LIN {X 0,Y 122.91,Z 344.93,A -85,B 0,C 180,E1 -26212.698,E2 -26212.698} C_VEL
LIN {X 0,Y 127.264,Z 335.4,A -85,B 0,C 180,E1 -26216.213,E2 -26216.213} C_VEL
LIN {X 0,Y 131.785,Z 325.121,A -85,B 0,C 180,E1 -26219.114,E2 -26219.114} C_VEL
LIN {X 0,Y 136.511,Z 312.597,A -85,B 0,C 180,E1 -26221.845,E2 -26221.845} C_VEL
LIN {X 0,Y 140.339,Z 300.53,A -85,B 0,C 180,E1 -26223.852,E2 -26223.852} C_VEL
LIN {X 0,Y 143.644,Z 287.351,A -85,B 0,C 180,E1 -26225.516,E2 -26225.516} C_VEL
LIN {X 0,Y 146.296,Z 273.12,A -85,B 0,C 180,E1 -26226.793,E2 -26226.793} C_VEL
LIN {X 0,Y 148.096,Z 259.317,A -85,B 0,C 180,E1 -26227.549,E2 -26227.549} C_VEL
LIN {X 0,Y 152.361,Z 207.795,A -85,B 0,C 180,E1 -26229.457,E2 -26229.457} C_VEL
LIN {X 0,Y 147.363,Z 196.9,A -85,B 0,C 180,E1 -26232.578,E2 -26232.578} C_VEL
LIN {X 0,Y 142.317,Z 187.434,A -85,B 0,C 180,E1 -26236.042,E2 -26236.042} C_VEL
LIN {X 0,Y 138.298,Z 180.817,A -85,B 0,C 180,E1 -26239.137,E2 -26239.137} C_VEL
LIN {X 0,Y 134.118,Z 174.322,A -85,B 0,C 180,E1 -26242.853,E2 -26242.853} C_VEL
LIN {X 0,Y 130.981,Z 169.962,A -85,B 0,C 180,E1 -26246.076,E2 -26246.076} C_VEL
LIN {X 0,Y 128.411,Z 166.477,A -85,B 0,C 180,E1 -26249.154,E2 -26249.154} C_VEL
LIN {X 0,Y 127.763,Z 165.521,A -85,B 0,C 180,E1 -26250.031,E2 -26250.031} C_VEL
LIN {X 0,Y 125.309,Z 162.834,A -85,B 0,C 180,E1 -26253.6,E2 -26253.6} C_VEL
LIN {X 0,Y 124.174,Z 160.568,A -85,B 0,C 180,E1 -26255.787,E2 -26255.787} C_VEL
LIN {X 0,Y 121.255,Z 158.023,A -85,B 0,C 180,E1 -26262.732,E2 -26262.732} C_VEL
LIN {X 0,Y 120.363,Z 155.046,A -85,B 0,C 180,E1 -26268.375,E2 -26268.375} C_VEL
LIN {X 0,Y 120.599,Z 154.855,A -85,B 0,C 180,E1 -26276.67,E2 -26276.67} C_VEL
LIN {X 0,Y 120.863,Z 155.058,A -85,B 0,C 180,E1 -26278.137,E2 -26278.137} C_VEL
LIN {X 0,Y 121.622,Z 157.801,A -85,B 0,C 180,E1 -26281.874,E2 -26281.874} C_VEL
LIN {X 0,Y 123.928,Z 160.174,A -85,B 0,C 180,E1 -26287.341,E2 -26287.341} C_VEL
LIN {X 0,Y 124.584,Z 160.744,A -85,B 0,C 180,E1 -26288.526,E2 -26288.526} C_VEL
LIN {X 0,Y 126.362,Z 163.972,A -85,B 0,C 180,E1 -26291.642,E2 -26291.642} C_VEL
LIN {X 0,Y 128.449,Z 166.176,A -85,B 0,C 180,E1 -26294.466,E2 -26294.466} C_VEL
LIN {X 0,Y 131.151,Z 169.964,A -85,B 0,C 180,E1 -26297.718,E2 -26297.718} C_VEL
LIN {X 0,Y 135.213,Z 176.102,A -85,B 0,C 180,E1 -26301.831,E2 -26301.831} C_VEL
LIN {X 0,Y 137.802,Z 180.05,A -85,B 0,C 180,E1 -26304.089,E2 -26304.089} C_VEL
LIN {X 0,Y 142.126,Z 187.185,A -85,B 0,C 180,E1 -26307.455,E2 -26307.455} C_VEL
LIN {X 0,Y 145.883,Z 194.238,A -85,B 0,C 180,E1 -26310.095,E2 -26310.095} C_VEL
LIN {X 0,Y 150.285,Z 206.436,A -85,B 0,C 180,E1 -26313.156,E2 -26313.156} C_VEL
LIN {X 0,Y 152.175,Z 212.724,A -85,B 0,C 180,E1 -26314.44,E2 -26314.44} C_VEL
LIN {X 0,Y 147.482,Z 269.48,A -85,B 0,C 180,E1 -26316.622,E2 -26316.622} C_VEL
LIN {X 0,Y 145.239,Z 284.153,A -85,B 0,C 180,E1 -26317.599,E2 -26317.599} C_VEL
LIN {X 0,Y 142.244,Z 297.61,A -85,B 0,C 180,E1 -26318.913,E2 -26318.913} C_VEL
LIN {X 0,Y 138.11,Z 311.658,A -85,B 0,C 180,E1 -26320.811,E2 -26320.811} C_VEL
LIN {X 0,Y 133.642,Z 324.22,A -85,B 0,C 180,E1 -26323.141,E2 -26323.141} C_VEL
LIN {X 0,Y 129.478,Z 334.557,A -85,B 0,C 180,E1 -26325.672,E2 -26325.672} C_VEL
LIN {X 0,Y 126.048,Z 342.338,A -85,B 0,C 180,E1 -26328.01,E2 -26328.01} C_VEL
LIN {X 0,Y 120.56,Z 353.468,A -85,B 0,C 180,E1 -26332.265,E2 -26332.265} C_VEL
LIN {X 0,Y 115.908,Z 362.657,A -85,B 0,C 180,E1 -26336.933,E2 -26336.933} C_VEL
LIN {X 0,Y 111.861,Z 370.547,A -85,B 0,C 180,E1 -26342.134,E2 -26342.134} C_VEL
LIN {X 0,Y 109.064,Z 376.625,A -85,B 0,C 180,E1 -26347.261,E2 -26347.261} C_VEL
LIN {X 0,Y 106.869,Z 381.829,A -85,B 0,C 180,E1 -26352.792,E2 -26352.792} C_VEL
LIN {X 0,Y 105.627,Z 386.001,A -85,B 0,C 180,E1 -26358.492,E2 -26358.492} C_VEL
LIN {X 0,Y 105.224,Z 388.285,A -85,B 0,C 180,E1 -26362.329,E2 -26362.329} C_VEL
LIN {X 0,Y 105.192,Z 391.7,A -85,B 0,C 180,E1 -26370.005,E2 -26370.005} C_VEL
LIN {X 0,Y 105.119,Z 392.843,A -85,B 0,C 180,E1 -26373.839,E2 -26373.839} C_VEL
LIN {X 0,Y 105.704,Z 394.109,A -85,B 0,C 180,E1 -26381.511,E2 -26381.511} C_VEL
LIN {X 0,Y 107.789,Z 394.075,A -85,B 0,C 180,E1 -26389.032,E2 -26389.032} C_VEL
LIN {X 0,Y 111.681,Z 392.762,A -85,B 0,C 180,E1 -26396.141,E2 -26396.141} C_VEL
LIN {X 0,Y 117.55,Z 389.878,A -85,B 0,C 180,E1 -26403.156,E2 -26403.156} C_VEL
LIN {X 0,Y 124.607,Z 385.667,A -85,B 0,C 180,E1 -26409.133,E2 -26409.133} C_VEL
LIN {X 0,Y 127.11,Z 383.713,A -85,B 0,C 180,E1 -26411.4,E2 -26411.4} C_VEL
LIN {X 0,Y 130.128,Z 380.241,A -85,B 0,C 180,E1 -26415.325,E2 -26415.325} C_VEL
LIN {X 0,Y 133.645,Z 376.307,A -85,B 0,C 180,E1 -26418.957,E2 -26418.957} C_VEL
LIN {X 0,Y 136.795,Z 373.532,A -85,B 0,C 180,E1 -26420.71,E2 -26420.71} C_VEL
LIN {X 0,Y 145.544,Z 366.023,A -85,B 0,C 180,E1 -26423.987,E2 -26423.987} C_VEL
LIN {X 0,Y 154.63,Z 356.799,A -85,B 0,C 180,E1 -26426.995,E2 -26426.995} C_VEL
LIN {X 0,Y 163.449,Z 346.525,A -85,B 0,C 180,E1 -26429.319,E2 -26429.319} C_VEL
LIN {X 0,Y 171.439,Z 335.446,A -85,B 0,C 180,E1 -26431.199,E2 -26431.199} C_VEL
LIN {X 0,Y 178.13,Z 324.469,A -85,B 0,C 180,E1 -26432.595,E2 -26432.595} C_VEL
LIN {X 0,Y 184.22,Z 312.561,A -85,B 0,C 180,E1 -26433.711,E2 -26433.711} C_VEL
LIN {X 0,Y 189.587,Z 299.462,A -85,B 0,C 180,E1 -26434.639,E2 -26434.639} C_VEL
LIN {X 0,Y 193.841,Z 285.948,A -85,B 0,C 180,E1 -26435.335,E2 -26435.335} C_VEL
LIN {X 0,Y 196.748,Z 273.12,A -85,B 0,C 180,E1 -26435.823,E2 -26435.823} C_VEL
LIN {X 0,Y 198.976,Z 257.031,A -85,B 0,C 180,E1 -26436.23,E2 -26436.23} C_VEL
LIN {X 0,Y 199.287,Z 253.75,A -85,B 0,C 180,E1 -26436.344,E2 -26436.344} C_VEL
LIN {X 0,Y 197.239,Z 247.184,A -85,B 0,C 180,E1 -26439.469,E2 -26439.469} C_VEL
LIN {X 0,Y 195.601,Z 242.329,A -85,B 0,C 180,E1 -26442.751,E2 -26442.751} C_VEL
LIN {X 0,Y 194.612,Z 239.828,A -85,B 0,C 180,E1 -26445.351,E2 -26445.351} C_VEL
LIN {X 0,Y 193.533,Z 236.708,A -85,B 0,C 180,E1 -26451.641,E2 -26451.641} C_VEL
LIN {X 0,Y 193.655,Z 236.699,A -85,B 0,C 180,E1 -26454.175,E2 -26454.175} C_VEL
LIN {X 0,Y 194.972,Z 240.283,A -85,B 0,C 180,E1 -26459.993,E2 -26459.993} C_VEL
LIN {X 0,Y 196.407,Z 243.777,A -85,B 0,C 180,E1 -26463.231,E2 -26463.231} C_VEL
LIN {X 0,Y 198.463,Z 248.409,A -85,B 0,C 180,E1 -26466.533,E2 -26466.533} C_VEL
LIN {X 0,Y 199.53,Z 250.985,A -85,B 0,C 180,E1 -26467.963,E2 -26467.963} C_VEL
LIN {X 0,Y 197.309,Z 268.548,A -85,B 0,C 180,E1 -26468.468,E2 -26468.468} C_VEL
LIN {X 0,Y 194.201,Z 282.697,A -85,B 0,C 180,E1 -26469.023,E2 -26469.023} C_VEL
LIN {X 0,Y 190.293,Z 295.304,A -85,B 0,C 180,E1 -26469.708,E2 -26469.708} C_VEL
LIN {X 0,Y 185.136,Z 308.381,A -85,B 0,C 180,E1 -26470.747,E2 -26470.747} C_VEL
LIN {X 0,Y 178.784,Z 321.146,A -85,B 0,C 180,E1 -26472.071,E2 -26472.071} C_VEL
LIN {X 0,Y 171.822,Z 332.609,A -85,B 0,C 180,E1 -26473.651,E2 -26473.651} C_VEL
LIN {X 0,Y 164.142,Z 343.196,A -85,B 0,C 180,E1 -26475.544,E2 -26475.544} C_VEL
LIN {X 0,Y 156.716,Z 352.027,A -85,B 0,C 180,E1 -26477.632,E2 -26477.632} C_VEL
LIN {X 0,Y 148.104,Z 360.827,A -85,B 0,C 180,E1 -26480.404,E2 -26480.404} C_VEL
LIN {X 0,Y 139.155,Z 368.672,A -85,B 0,C 180,E1 -26483.82,E2 -26483.82} C_VEL
LIN {X 0,Y 130.895,Z 374.913,A -85,B 0,C 180,E1 -26487.627,E2 -26487.627} C_VEL
LIN {X 0,Y 123.838,Z 379.589,A -85,B 0,C 180,E1 -26491.641,E2 -26491.641} C_VEL
LIN {X 0,Y 115.676,Z 384.074,A -85,B 0,C 180,E1 -26497.397,E2 -26497.397} C_VEL
LIN {X 0,Y 108.425,Z 387.236,A -85,B 0,C 180,E1 -26504.513,E2 -26504.513} C_VEL
LIN {X 0,Y 103.082,Z 388.764,A -85,B 0,C 180,E1 -26512.142,E2 -26512.142} C_VEL
LIN {X 0,Y 99.548,Z 388.842,A -85,B 0,C 180,E1 -26520.377,E2 -26520.377} C_VEL
LIN {X 0,Y 97.829,Z 387.459,A -85,B 0,C 180,E1 -26529.011,E2 -26529.011} C_VEL
LIN {X 0,Y 97.525,Z 386.246,A -85,B 0,C 180,E1 -26533.241,E2 -26533.241} C_VEL
LIN {X 0,Y 98.023,Z 382.697,A -85,B 0,C 180,E1 -26541.75,E2 -26541.75} C_VEL
LIN {X 0,Y 99.346,Z 379.08,A -85,B 0,C 180,E1 -26547.967,E2 -26547.967} C_VEL
LIN {X 0,Y 101.284,Z 374.503,A -85,B 0,C 180,E1 -26553.973,E2 -26553.973} C_VEL
LIN {X 0,Y 104.649,Z 367.913,A -85,B 0,C 180,E1 -26560.637,E2 -26560.637} C_VEL
LIN {X 0,Y 109.179,Z 359.737,A -85,B 0,C 180,E1 -26566.833,E2 -26566.833} C_VEL
LIN {X 0,Y 113.83,Z 351.181,A -85,B 0,C 180,E1 -26571.738,E2 -26571.738} C_VEL
LIN {X 0,Y 118.098,Z 342.71,A -85,B 0,C 180,E1 -26575.554,E2 -26575.554} C_VEL
LIN {X 0,Y 122.512,Z 333.725,A -85,B 0,C 180,E1 -26578.709,E2 -26578.709} C_VEL
LIN {X 0,Y 127.733,Z 321.8,A -85,B 0,C 180,E1 -26581.971,E2 -26581.971} C_VEL
LIN {X 0,Y 132.219,Z 310.069,A -85,B 0,C 180,E1 -26584.38,E2 -26584.38} C_VEL
LIN {X 0,Y 136.535,Z 296.316,A -85,B 0,C 180,E1 -26586.519,E2 -26586.519} C_VEL
LIN {X 0,Y 139.845,Z 282.308,A -85,B 0,C 180,E1 -26588.107,E2 -26588.107} C_VEL
LIN {X 0,Y 142.238,Z 268.536,A -85,B 0,C 180,E1 -26589.157,E2 -26589.157} C_VEL
LIN {X 0,Y 144.089,Z 251.322,A -85,B 0,C 180,E1 -26589.922,E2 -26589.922} C_VEL
LIN {X 0,Y 147.539,Z 210.291,A -85,B 0,C 180,E1 -26591.453,E2 -26591.453} C_VEL
LIN {X 0,Y 143.283,Z 200.805,A -85,B 0,C 180,E1 -26594.355,E2 -26594.355} C_VEL
LIN {X 0,Y 138.513,Z 191.636,A -85,B 0,C 180,E1 -26597.951,E2 -26597.951} C_VEL
LIN {X 0,Y 135.152,Z 185.928,A -85,B 0,C 180,E1 -26600.799,E2 -26600.799} C_VEL
LIN {X 0,Y 131.35,Z 179.866,A -85,B 0,C 180,E1 -26604.502,E2 -26604.502} C_VEL
LIN {X 0,Y 128.942,Z 176.298,A -85,B 0,C 180,E1 -26607.199,E2 -26607.199} C_VEL
LIN {X 0,Y 125.898,Z 171.998,A -85,B 0,C 180,E1 -26611.214,E2 -26611.214} C_VEL
LIN {X 0,Y 123.5,Z 168.944,A -85,B 0,C 180,E1 -26615.11,E2 -26615.11} C_VEL
LIN {X 0,Y 122.683,Z 167.345,A -85,B 0,C 180,E1 -26616.827,E2 -26616.827} C_VEL
LIN {X 0,Y 120.011,Z 164.606,A -85,B 0,C 180,E1 -26624.079,E2 -26624.079} C_VEL
LIN {X 0,Y 119.42,Z 162.041,A -85,B 0,C 180,E1 -26628.958,E2 -26628.958} C_VEL
LIN {X 0,Y 119.78,Z 161.905,A -85,B 0,C 180,E1 -26637.068,E2 -26637.068} C_VEL
LIN {X 0,Y 120.765,Z 165.154,A -85,B 0,C 180,E1 -26642.095,E2 -26642.095} C_VEL
LIN {X 0,Y 123.12,Z 167.53,A -85,B 0,C 180,E1 -26647.596,E2 -26647.596} C_VEL
LIN {X 0,Y 125.06,Z 170.939,A -85,B 0,C 180,E1 -26651.149,E2 -26651.149} C_VEL
LIN {X 0,Y 126.635,Z 172.708,A -85,B 0,C 180,E1 -26653.41,E2 -26653.41} C_VEL
LIN {X 0,Y 129.754,Z 177.467,A -85,B 0,C 180,E1 -26657.382,E2 -26657.382} C_VEL
LIN {X 0,Y 132.774,Z 182.144,A -85,B 0,C 180,E1 -26660.602,E2 -26660.602} C_VEL
LIN {X 0,Y 136.308,Z 187.774,A -85,B 0,C 180,E1 -26663.845,E2 -26663.845} C_VEL
LIN {X 0,Y 141.473,Z 197.254,A -85,B 0,C 180,E1 -26667.968,E2 -26667.968} C_VEL
LIN {X 0,Y 144.23,Z 204.494,A -85,B 0,C 180,E1 -26670.074,E2 -26670.074} C_VEL
LIN {X 0,Y 147.292,Z 214.306,A -85,B 0,C 180,E1 -26672.371,E2 -26672.371} C_VEL
LIN {X 0,Y 147.076,Z 218.929,A -85,B 0,C 180,E1 -26672.622,E2 -26672.622} C_VEL
LIN {X 0,Y 142.67,Z 269.478,A -85,B 0,C 180,E1 -26674.564,E2 -26674.564} C_VEL
LIN {X 0,Y 140.345,Z 284.092,A -85,B 0,C 180,E1 -26675.544,E2 -26675.544} C_VEL
LIN {X 0,Y 137.234,Z 297.516,A -85,B 0,C 180,E1 -26676.86,E2 -26676.86} C_VEL
LIN {X 0,Y 132.937,Z 311.543,A -85,B 0,C 180,E1 -26678.766,E2 -26678.766} C_VEL
LIN {X 0,Y 128.231,Z 324.184,A -85,B 0,C 180,E1 -26681.136,E2 -26681.136} C_VEL
LIN {X 0,Y 123.909,Z 334.415,A -85,B 0,C 180,E1 -26683.69,E2 -26683.69} C_VEL
LIN {X 0,Y 120.296,Z 342.186,A -85,B 0,C 180,E1 -26686.078,E2 -26686.078} C_VEL
LIN {X 0,Y 114.956,Z 352.48,A -85,B 0,C 180,E1 -26690.071,E2 -26690.071} C_VEL
LIN {X 0,Y 109.973,Z 361.805,A -85,B 0,C 180,E1 -26694.896,E2 -26694.896} C_VEL
LIN {X 0,Y 105.756,Z 369.452,A -85,B 0,C 180,E1 -26700.028,E2 -26700.028} C_VEL
LIN {X 0,Y 102.466,Z 375.984,A -85,B 0,C 180,E1 -26705.705,E2 -26705.705} C_VEL
LIN {X 0,Y 100.041,Z 381.241,A -85,B 0,C 180,E1 -26711.577,E2 -26711.577} C_VEL
LIN {X 0,Y 98.642,Z 385.505,A -85,B 0,C 180,E1 -26717.664,E2 -26717.664} C_VEL
LIN {X 0,Y 98.176,Z 387.834,A -85,B 0,C 180,E1 -26721.775,E2 -26721.775} C_VEL
LIN {X 0,Y 98.096,Z 391.33,A -85,B 0,C 180,E1 -26730.006,E2 -26730.006} C_VEL
LIN {X 0,Y 98.029,Z 392.512,A -85,B 0,C 180,E1 -26734.117,E2 -26734.117} C_VEL
LIN {X 0,Y 98.727,Z 393.855,A -85,B 0,C 180,E1 -26742.337,E2 -26742.337} C_VEL
LIN {X 0,Y 101.062,Z 393.897,A -85,B 0,C 180,E1 -26750.353,E2 -26750.353} C_VEL
LIN {X 0,Y 105.312,Z 392.666,A -85,B 0,C 180,E1 -26757.855,E2 -26757.855} C_VEL
LIN {X 0,Y 111.235,Z 390.106,A -85,B 0,C 180,E1 -26764.761,E2 -26764.761} C_VEL
LIN {X 0,Y 118.783,Z 386.019,A -85,B 0,C 180,E1 -26771.03,E2 -26771.03} C_VEL
LIN {X 0,Y 126.949,Z 380.85,A -85,B 0,C 180,E1 -26776.035,E2 -26776.035} C_VEL
LIN {X 0,Y 133.996,Z 375.737,A -85,B 0,C 180,E1 -26779.516,E2 -26779.516} C_VEL
LIN {X 0,Y 136.795,Z 373.532,A -85,B 0,C 180,E1 -26780.71,E2 -26780.71} C_VEL
LIN {X 0,Y 140.018,Z 370.602,A -85,B 0,C 180,E1 -26782.367,E2 -26782.367} C_VEL
LIN {X 0,Y 144.128,Z 365.614,A -85,B 0,C 180,E1 -26785.422,E2 -26785.422} C_VEL
LIN {X 0,Y 148.389,Z 360.232,A -85,B 0,C 180,E1 -26788.219,E2 -26788.219} C_VEL
LIN {X 0,Y 151.717,Z 356.53,A -85,B 0,C 180,E1 -26789.454,E2 -26789.454} C_VEL
LIN {X 0,Y 159.964,Z 347.236,A -85,B 0,C 180,E1 -26791.493,E2 -26791.493} C_VEL
LIN {X 0,Y 168.165,Z 336.357,A -85,B 0,C 180,E1 -26793.299,E2 -26793.299} C_VEL
LIN {X 0,Y 175.001,Z 325.599,A -85,B 0,C 180,E1 -26794.641,E2 -26794.641} C_VEL
LIN {X 0,Y 181.218,Z 313.993,A -85,B 0,C 180,E1 -26795.703,E2 -26795.703} C_VEL
LIN {X 0,Y 186.677,Z 301.395,A -85,B 0,C 180,E1 -26796.594,E2 -26796.594} C_VEL
LIN {X 0,Y 191.059,Z 288.5,A -85,B 0,C 180,E1 -26797.248,E2 -26797.248} C_VEL
LIN {X 0,Y 194.33,Z 275.303,A -85,B 0,C 180,E1 -26797.755,E2 -26797.755} C_VEL
LIN {X 0,Y 196.703,Z 260.3,A -85,B 0,C 180,E1 -26798.127,E2 -26798.127} C_VEL
LIN {X 0,Y 196.932,Z 257.596,A -85,B 0,C 180,E1 -26798.261,E2 -26798.261} C_VEL
LIN {X 0,Y 195.511,Z 252.638,A -85,B 0,C 180,E1 -26800.84,E2 -26800.84} C_VEL
LIN {X 0,Y 194.366,Z 248.965,A -85,B 0,C 180,E1 -26803.45,E2 -26803.45} C_VEL
LIN {X 0,Y 193.551,Z 246.75,A -85,B 0,C 180,E1 -26805.806,E2 -26805.806} C_VEL
LIN {X 0,Y 192.64,Z 243.839,A -85,B 0,C 180,E1 -26811.602,E2 -26811.602} C_VEL
LIN {X 0,Y 192.762,Z 243.785,A -85,B 0,C 180,E1 -26814.148,E2 -26814.148} C_VEL
LIN {X 0,Y 193.91,Z 247.232,A -85,B 0,C 180,E1 -26819.604,E2 -26819.604} C_VEL
LIN {X 0,Y 195.252,Z 250.712,A -85,B 0,C 180,E1 -26822.83,E2 -26822.83} C_VEL
LIN {X 0,Y 197.001,Z 254.991,A -85,B 0,C 180,E1 -26825.861,E2 -26825.861} C_VEL
LIN {X 0,Y 197.173,Z 255.516,A -85,B 0,C 180,E1 -26826.131,E2 -26826.131} C_VEL
LIN {X 0,Y 194.888,Z 271.328,A -85,B 0,C 180,E1 -26826.571,E2 -26826.571} C_VEL
LIN {X 0,Y 191.611,Z 284.922,A -85,B 0,C 180,E1 -26827.096,E2 -26827.096} C_VEL
LIN {X 0,Y 187.534,Z 297.324,A -85,B 0,C 180,E1 -26827.773,E2 -26827.773} C_VEL
LIN {X 0,Y 182.058,Z 310.391,A -85,B 0,C 180,E1 -26828.807,E2 -26828.807} C_VEL
LIN {X 0,Y 175.76,Z 322.398,A -85,B 0,C 180,E1 -26830.03,E2 -26830.03} C_VEL
LIN {X 0,Y 168.584,Z 333.727,A -85,B 0,C 180,E1 -26831.556,E2 -26831.556} C_VEL
LIN {X 0,Y 160.739,Z 344.111,A -85,B 0,C 180,E1 -26833.371,E2 -26833.371} C_VEL
LIN {X 0,Y 153.089,Z 352.823,A -85,B 0,C 180,E1 -26835.393,E2 -26835.393} C_VEL
LIN {X 0,Y 144.186,Z 361.518,A -85,B 0,C 180,E1 -26838.095,E2 -26838.095} C_VEL
LIN {X 0,Y 135.243,Z 369.009,A -85,B 0,C 180,E1 -26841.32,E2 -26841.32} C_VEL
LIN {X 0,Y 127.562,Z 374.594,A -85,B 0,C 180,E1 -26844.614,E2 -26844.614} C_VEL
LIN {X 0,Y 120.031,Z 379.342,A -85,B 0,C 180,E1 -26848.556,E2 -26848.556} C_VEL
LIN {X 0,Y 113.068,Z 383.068,A -85,B 0,C 180,E1 -26852.944,E2 -26852.944} C_VEL
LIN {X 0,Y 106.875,Z 385.886,A -85,B 0,C 180,E1 -26857.889,E2 -26857.889} C_VEL
LIN {X 0,Y 99.994,Z 388.261,A -85,B 0,C 180,E1 -26865.337,E2 -26865.337} C_VEL
LIN {X 0,Y 94.911,Z 389.164,A -85,B 0,C 180,E1 -26873.666,E2 -26873.666} C_VEL
LIN {X 0,Y 91.732,Z 388.629,A -85,B 0,C 180,E1 -26882.626,E2 -26882.626} C_VEL
LIN {X 0,Y 90.783,Z 387.614,A -85,B 0,C 180,E1 -26888.233,E2 -26888.233} C_VEL
LIN {X 0,Y 90.401,Z 385.149,A -85,B 0,C 180,E1 -26896.506,E2 -26896.506} C_VEL
LIN {X 0,Y 91.628,Z 380.96,A -85,B 0,C 180,E1 -26905.595,E2 -26905.595} C_VEL
LIN {X 0,Y 93.362,Z 376.841,A -85,B 0,C 180,E1 -26912.151,E2 -26912.151} C_VEL
LIN {X 0,Y 95.921,Z 371.716,A -85,B 0,C 180,E1 -26918.42,E2 -26918.42} C_VEL
LIN {X 0,Y 100.204,Z 364.386,A -85,B 0,C 180,E1 -26925.243,E2 -26925.243} C_VEL
LIN {X 0,Y 105.04,Z 356.234,A -85,B 0,C 180,E1 -26930.915,E2 -26930.915} C_VEL
LIN {X 0,Y 109.98,Z 347.504,A -85,B 0,C 180,E1 -26935.547,E2 -26935.547} C_VEL
LIN {X 0,Y 115.154,Z 337.389,A -85,B 0,C 180,E1 -26939.722,E2 -26939.722} C_VEL
LIN {X 0,Y 120.652,Z 326.189,A -85,B 0,C 180,E1 -26943.093,E2 -26943.093} C_VEL
LIN {X 0,Y 125.829,Z 313.831,A -85,B 0,C 180,E1 -26945.9,E2 -26945.9} C_VEL
LIN {X 0,Y 129.99,Z 301.974,A -85,B 0,C 180,E1 -26947.946,E2 -26947.946} C_VEL
LIN {X 0,Y 133.58,Z 289.111,A -85,B 0,C 180,E1 -26949.632,E2 -26949.632} C_VEL
LIN {X 0,Y 136.65,Z 274.481,A -85,B 0,C 180,E1 -26950.97,E2 -26950.97} C_VEL
LIN {X 0,Y 138.657,Z 260.38,A -85,B 0,C 180,E1 -26951.775,E2 -26951.775} C_VEL
LIN {X 0,Y 142.916,Z 212.87,A -85,B 0,C 180,E1 -26953.544,E2 -26953.544} C_VEL
LIN {X 0,Y 138.94,Z 203.896,A -85,B 0,C 180,E1 -26956.546,E2 -26956.546} C_VEL
LIN {X 0,Y 134.376,Z 194.924,A -85,B 0,C 180,E1 -26960.411,E2 -26960.411} C_VEL
LIN {X 0,Y 129.944,Z 187.265,A -85,B 0,C 180,E1 -26964.826,E2 -26964.826} C_VEL
LIN {X 0,Y 126.936,Z 182.619,A -85,B 0,C 180,E1 -26968.378,E2 -26968.378} C_VEL
LIN {X 0,Y 124.256,Z 178.611,A -85,B 0,C 180,E1 -26972.186,E2 -26972.186} C_VEL
LIN {X 0,Y 121.836,Z 175.161,A -85,B 0,C 180,E1 -26976.527,E2 -26976.527} C_VEL
LIN {X 0,Y 121.406,Z 174.223,A -85,B 0,C 180,E1 -26977.53,E2 -26977.53} C_VEL
LIN {X 0,Y 118.84,Z 171.148,A -85,B 0,C 180,E1 -26985.455,E2 -26985.455} C_VEL
LIN {X 0,Y 118.483,Z 168.952,A -85,B 0,C 180,E1 -26989.761,E2 -26989.761} C_VEL
LIN {X 0,Y 118.825,Z 169.057,A -85,B 0,C 180,E1 -26996.774,E2 -26996.774} C_VEL
LIN {X 0,Y 119.66,Z 172.036,A -85,B 0,C 180,E1 -27001.464,E2 -27001.464} C_VEL
LIN {X 0,Y 121.74,Z 174.355,A -85,B 0,C 180,E1 -27006.745,E2 -27006.745} C_VEL
LIN {X 0,Y 123.649,Z 177.74,A -85,B 0,C 180,E1 -27010.449,E2 -27010.449} C_VEL
LIN {X 0,Y 125.043,Z 179.504,A -85,B 0,C 180,E1 -27012.59,E2 -27012.59} C_VEL
LIN {X 0,Y 127.779,Z 183.879,A -85,B 0,C 180,E1 -27016.309,E2 -27016.309} C_VEL
LIN {X 0,Y 130.599,Z 188.472,A -85,B 0,C 180,E1 -27019.536,E2 -27019.536} C_VEL
LIN {X 0,Y 133.937,Z 194.178,A -85,B 0,C 180,E1 -27022.826,E2 -27022.826} C_VEL
LIN {X 0,Y 138.497,Z 203.038,A -85,B 0,C 180,E1 -27026.738,E2 -27026.738} C_VEL
LIN {X 0,Y 142.194,Z 214.454,A -85,B 0,C 180,E1 -27029.834,E2 -27029.834} C_VEL
LIN {X 0,Y 142.784,Z 216.463,A -85,B 0,C 180,E1 -27030.309,E2 -27030.309} C_VEL
LIN {X 0,Y 138.178,Z 268.485,A -85,B 0,C 180,E1 -27032.322,E2 -27032.322} C_VEL
LIN {X 0,Y 135.854,Z 282.883,A -85,B 0,C 180,E1 -27033.246,E2 -27033.246} C_VEL
LIN {X 0,Y 132.76,Z 296.243,A -85,B 0,C 180,E1 -27034.537,E2 -27034.537} C_VEL
LIN {X 0,Y 128.602,Z 309.618,A -85,B 0,C 180,E1 -27036.294,E2 -27036.294} C_VEL
LIN {X 0,Y 124.162,Z 321.339,A -85,B 0,C 180,E1 -27038.377,E2 -27038.377} C_VEL
LIN {X 0,Y 119.114,Z 333.08,A -85,B 0,C 180,E1 -27041.22,E2 -27041.22} C_VEL
LIN {X 0,Y 115.182,Z 340.964,A -85,B 0,C 180,E1 -27043.575,E2 -27043.575} C_VEL
LIN {X 0,Y 109.555,Z 351.478,A -85,B 0,C 180,E1 -27047.663,E2 -27047.663} C_VEL
LIN {X 0,Y 104.168,Z 360.949,A -85,B 0,C 180,E1 -27052.619,E2 -27052.619} C_VEL
LIN {X 0,Y 99.201,Z 369.362,A -85,B 0,C 180,E1 -27058.502,E2 -27058.502} C_VEL
LIN {X 0,Y 95.955,Z 375.307,A -85,B 0,C 180,E1 -27063.938,E2 -27063.938} C_VEL
LIN {X 0,Y 93.279,Z 380.654,A -85,B 0,C 180,E1 -27070.188,E2 -27070.188} C_VEL
LIN {X 0,Y 91.354,Z 386.266,A -85,B 0,C 180,E1 -27078.918,E2 -27078.918} C_VEL
LIN {X 0,Y 90.886,Z 389.358,A -85,B 0,C 180,E1 -27085.571,E2 -27085.571} C_VEL
LIN {X 0,Y 90.993,Z 390.961,A -85,B 0,C 180,E1 -27090.006,E2 -27090.006} C_VEL
LIN {X 0,Y 90.936,Z 392.18,A -85,B 0,C 180,E1 -27094.439,E2 -27094.439} C_VEL
LIN {X 0,Y 91.783,Z 393.599,A -85,B 0,C 180,E1 -27103.287,E2 -27103.287} C_VEL
LIN {X 0,Y 94.396,Z 393.721,A -85,B 0,C 180,E1 -27111.862,E2 -27111.862} C_VEL
LIN {X 0,Y 99.051,Z 392.572,A -85,B 0,C 180,E1 -27119.787,E2 -27119.787} C_VEL
LIN {X 0,Y 105.375,Z 390.129,A -85,B 0,C 180,E1 -27126.895,E2 -27126.895} C_VEL
LIN {X 0,Y 113.114,Z 386.332,A -85,B 0,C 180,E1 -27133.121,E2 -27133.121} C_VEL
LIN {X 0,Y 122.11,Z 381.063,A -85,B 0,C 180,E1 -27138.442,E2 -27138.442} C_VEL
LIN {X 0,Y 129.499,Z 376.004,A -85,B 0,C 180,E1 -27141.906,E2 -27141.906} C_VEL
LIN {X 0,Y 138.766,Z 368.815,A -85,B 0,C 180,E1 -27145.394,E2 -27145.394} C_VEL
LIN {X 0,Y 147.442,Z 360.885,A -85,B 0,C 180,E1 -27148.223,E2 -27148.223} C_VEL
LIN {X 0,Y 151.717,Z 356.53,A -85,B 0,C 180,E1 -27149.454,E2 -27149.454} C_VEL
LIN {X 0,Y 155.06,Z 352.734,A -85,B 0,C 180,E1 -27150.605,E2 -27150.605} C_VEL
LIN {X 0,Y 159.487,Z 346.414,A -85,B 0,C 180,E1 -27152.89,E2 -27152.89} C_VEL
LIN {X 0,Y 163.722,Z 339.623,A -85,B 0,C 180,E1 -27154.968,E2 -27154.968} C_VEL
LIN {X 0,Y 166.653,Z 335.096,A -85,B 0,C 180,E1 -27155.802,E2 -27155.802} C_VEL
LIN {X 0,Y 174.47,Z 322.746,A -85,B 0,C 180,E1 -27157.146,E2 -27157.146} C_VEL
LIN {X 0,Y 180.831,Z 310.513,A -85,B 0,C 180,E1 -27158.118,E2 -27158.118} C_VEL
LIN {X 0,Y 186.401,Z 296.966,A -85,B 0,C 180,E1 -27158.941,E2 -27158.941} C_VEL
LIN {X 0,Y 190.773,Z 283.019,A -85,B 0,C 180,E1 -27159.509,E2 -27159.509} C_VEL
LIN {X 0,Y 193.711,Z 269.415,A -85,B 0,C 180,E1 -27159.94,E2 -27159.94} C_VEL
LIN {X 0,Y 194.819,Z 261.782,A -85,B 0,C 180,E1 -27160.143,E2 -27160.143} C_VEL
LIN {X 0,Y 193.961,Z 258.48,A -85,B 0,C 180,E1 -27162.055,E2 -27162.055} C_VEL
LIN {X 0,Y 193.163,Z 255.576,A -85,B 0,C 180,E1 -27164.158,E2 -27164.158} C_VEL
LIN {X 0,Y 192.508,Z 253.629,A -85,B 0,C 180,E1 -27166.266,E2 -27166.266} C_VEL
LIN {X 0,Y 191.748,Z 250.817,A -85,B 0,C 180,E1 -27172.079,E2 -27172.079} C_VEL
LIN {X 0,Y 191.865,Z 250.893,A -85,B 0,C 180,E1 -27174.121,E2 -27174.121} C_VEL
LIN {X 0,Y 192.861,Z 254.147,A -85,B 0,C 180,E1 -27179.21,E2 -27179.21} C_VEL
LIN {X 0,Y 193.944,Z 257.216,A -85,B 0,C 180,E1 -27182.07,E2 -27182.07} C_VEL
LIN {X 0,Y 194.983,Z 260.105,A -85,B 0,C 180,E1 -27184.224,E2 -27184.224} C_VEL
LIN {X 0,Y 192.475,Z 274.658,A -85,B 0,C 180,E1 -27184.643,E2 -27184.643} C_VEL
LIN {X 0,Y 188.71,Z 288.649,A -85,B 0,C 180,E1 -27185.187,E2 -27185.187} C_VEL
LIN {X 0,Y 183.732,Z 302.273,A -85,B 0,C 180,E1 -27185.968,E2 -27185.968} C_VEL
LIN {X 0,Y 177.805,Z 315.057,A -85,B 0,C 180,E1 -27187.04,E2 -27187.04} C_VEL
LIN {X 0,Y 170.505,Z 327.639,A -85,B 0,C 180,E1 -27188.388,E2 -27188.388} C_VEL
LIN {X 0,Y 162.912,Z 338.454,A -85,B 0,C 180,E1 -27189.928,E2 -27189.928} C_VEL
LIN {X 0,Y 154.398,Z 348.646,A -85,B 0,C 180,E1 -27191.844,E2 -27191.844} C_VEL
LIN {X 0,Y 145.089,Z 358.126,A -85,B 0,C 180,E1 -27194.339,E2 -27194.339} C_VEL
LIN {X 0,Y 136.046,Z 365.924,A -85,B 0,C 180,E1 -27197.107,E2 -27197.107} C_VEL
LIN {X 0,Y 127.395,Z 372.351,A -85,B 0,C 180,E1 -27200.296,E2 -27200.296} C_VEL
LIN {X 0,Y 117.697,Z 378.451,A -85,B 0,C 180,E1 -27204.694,E2 -27204.694} C_VEL
LIN {X 0,Y 109.13,Z 382.928,A -85,B 0,C 180,E1 -27209.601,E2 -27209.601} C_VEL
LIN {X 0,Y 102.383,Z 385.857,A -85,B 0,C 180,E1 -27214.53,E2 -27214.53} C_VEL
LIN {X 0,Y 94.746,Z 388.338,A -85,B 0,C 180,E1 -27222.108,E2 -27222.108} C_VEL
LIN {X 0,Y 88.916,Z 389.346,A -85,B 0,C 180,E1 -27230.77,E2 -27230.77} C_VEL
LIN {X 0,Y 85.122,Z 388.914,A -85,B 0,C 180,E1 -27240.297,E2 -27240.297} C_VEL
LIN {X 0,Y 83.796,Z 387.781,A -85,B 0,C 180,E1 -27247.26,E2 -27247.26} C_VEL
LIN {X 0,Y 83.261,Z 385.595,A -85,B 0,C 180,E1 -27255.324,E2 -27255.324} C_VEL
LIN {X 0,Y 83.914,Z 382.677,A -85,B 0,C 180,E1 -27262.776,E2 -27262.776} C_VEL
LIN {X 0,Y 85.491,Z 378.934,A -85,B 0,C 180,E1 -27269.993,E2 -27269.993} C_VEL
LIN {X 0,Y 87.85,Z 374.278,A -85,B 0,C 180,E1 -27276.886,E2 -27276.886} C_VEL
LIN {X 0,Y 91.896,Z 367.526,A -85,B 0,C 180,E1 -27284.385,E2 -27284.385} C_VEL
LIN {X 0,Y 97.257,Z 359.105,A -85,B 0,C 180,E1 -27291.174,E2 -27291.174} C_VEL
LIN {X 0,Y 102.664,Z 350.288,A -85,B 0,C 180,E1 -27296.447,E2 -27296.447} C_VEL
LIN {X 0,Y 108.485,Z 339.763,A -85,B 0,C 180,E1 -27301.209,E2 -27301.209} C_VEL
LIN {X 0,Y 114.23,Z 328.993,A -85,B 0,C 180,E1 -27304.682,E2 -27304.682} C_VEL
LIN {X 0,Y 119.509,Z 317.288,A -85,B 0,C 180,E1 -27307.592,E2 -27307.592} C_VEL
LIN {X 0,Y 124.446,Z 304.399,A -85,B 0,C 180,E1 -27309.964,E2 -27309.964} C_VEL
LIN {X 0,Y 128.517,Z 291.046,A -85,B 0,C 180,E1 -27311.789,E2 -27311.789} C_VEL
LIN {X 0,Y 131.74,Z 277.235,A -85,B 0,C 180,E1 -27313.113,E2 -27313.113} C_VEL
LIN {X 0,Y 133.778,Z 264.538,A -85,B 0,C 180,E1 -27313.943,E2 -27313.943} C_VEL
LIN {X 0,Y 138.442,Z 215.431,A -85,B 0,C 180,E1 -27315.794,E2 -27315.794} C_VEL
LIN {X 0,Y 134.276,Z 205.957,A -85,B 0,C 180,E1 -27319.34,E2 -27319.34} C_VEL
LIN {X 0,Y 130.738,Z 198.829,A -85,B 0,C 180,E1 -27322.758,E2 -27322.758} C_VEL
LIN {X 0,Y 126.925,Z 192.104,A -85,B 0,C 180,E1 -27327.045,E2 -27327.045} C_VEL
LIN {X 0,Y 124.835,Z 188.728,A -85,B 0,C 180,E1 -27329.801,E2 -27329.801} C_VEL
LIN {X 0,Y 122.643,Z 185.192,A -85,B 0,C 180,E1 -27333.2,E2 -27333.2} C_VEL
LIN {X 0,Y 120.394,Z 181.745,A -85,B 0,C 180,E1 -27337.599,E2 -27337.599} C_VEL
LIN {X 0,Y 119.969,Z 180.957,A -85,B 0,C 180,E1 -27338.65,E2 -27338.65} C_VEL
LIN {X 0,Y 117.766,Z 177.789,A -85,B 0,C 180,E1 -27346.628,E2 -27346.628} C_VEL
LIN {X 0,Y 117.576,Z 175.964,A -85,B 0,C 180,E1 -27350.165,E2 -27350.165} C_VEL
LIN {X 0,Y 117.838,Z 176.044,A -85,B 0,C 180,E1 -27356.112,E2 -27356.112} C_VEL
LIN {X 0,Y 118.657,Z 179.065,A -85,B 0,C 180,E1 -27361.148,E2 -27361.148} C_VEL
LIN {X 0,Y 120.35,Z 181.121,A -85,B 0,C 180,E1 -27365.787,E2 -27365.787} C_VEL
LIN {X 0,Y 122.373,Z 184.668,A -85,B 0,C 180,E1 -27369.932,E2 -27369.932} C_VEL
LIN {X 0,Y 123.513,Z 186.359,A -85,B 0,C 180,E1 -27371.81,E2 -27371.81} C_VEL
LIN {X 0,Y 125.806,Z 190.193,A -85,B 0,C 180,E1 -27375.139,E2 -27375.139} C_VEL
LIN {X 0,Y 129.328,Z 196.282,A -85,B 0,C 180,E1 -27379.387,E2 -27379.387} C_VEL
LIN {X 0,Y 132.888,Z 203.17,A -85,B 0,C 180,E1 -27383.016,E2 -27383.016} C_VEL
LIN {X 0,Y 135.32,Z 208.531,A -85,B 0,C 180,E1 -27385.252,E2 -27385.252} C_VEL
LIN {X 0,Y 138.37,Z 218.636,A -85,B 0,C 180,E1 -27388.08,E2 -27388.08} C_VEL
LIN {X 0,Y 133.719,Z 268.711,A -85,B 0,C 180,E1 -27390.006,E2 -27390.006} C_VEL
LIN {X 0,Y 131.262,Z 283.113,A -85,B 0,C 180,E1 -27390.929,E2 -27390.929} C_VEL
LIN {X 0,Y 127.804,Z 297.124,A -85,B 0,C 180,E1 -27392.286,E2 -27392.286} C_VEL
LIN {X 0,Y 123.163,Z 311.157,A -85,B 0,C 180,E1 -27394.175,E2 -27394.175} C_VEL
LIN {X 0,Y 118.013,Z 323.855,A -85,B 0,C 180,E1 -27396.563,E2 -27396.563} C_VEL
LIN {X 0,Y 113.28,Z 334.037,A -85,B 0,C 180,E1 -27399.157,E2 -27399.157} C_VEL
LIN {X 0,Y 109.261,Z 341.806,A -85,B 0,C 180,E1 -27401.612,E2 -27401.612} C_VEL
LIN {X 0,Y 103.33,Z 352.105,A -85,B 0,C 180,E1 -27405.809,E2 -27405.809} C_VEL
LIN {X 0,Y 97.66,Z 361.428,A -85,B 0,C 180,E1 -27410.981,E2 -27410.981} C_VEL
LIN {X 0,Y 92.728,Z 369.237,A -85,B 0,C 180,E1 -27416.762,E2 -27416.762} C_VEL
LIN {X 0,Y 89.562,Z 374.592,A -85,B 0,C 180,E1 -27421.919,E2 -27421.919} C_VEL
LIN {X 0,Y 86.591,Z 380.046,A -85,B 0,C 180,E1 -27428.585,E2 -27428.585} C_VEL
LIN {X 0,Y 84.346,Z 385.753,A -85,B 0,C 180,E1 -27437.984,E2 -27437.984} C_VEL
LIN {X 0,Y 83.801,Z 388.936,A -85,B 0,C 180,E1 -27445.196,E2 -27445.196} C_VEL
LIN {X 0,Y 83.9,Z 390.581,A -85,B 0,C 180,E1 -27450.007,E2 -27450.007} C_VEL
LIN {X 0,Y 83.867,Z 391.841,A -85,B 0,C 180,E1 -27454.814,E2 -27454.814} C_VEL
LIN {X 0,Y 84.863,Z 393.34,A -85,B 0,C 180,E1 -27464.392,E2 -27464.392} C_VEL
LIN {X 0,Y 87.809,Z 393.544,A -85,B 0,C 180,E1 -27473.597,E2 -27473.597} C_VEL
LIN {X 0,Y 92.922,Z 392.478,A -85,B 0,C 180,E1 -27481.974,E2 -27481.974} C_VEL
LIN {X 0,Y 99.758,Z 390.119,A -85,B 0,C 180,E1 -27489.357,E2 -27489.357} C_VEL
LIN {X 0,Y 108.015,Z 386.409,A -85,B 0,C 180,E1 -27495.709,E2 -27495.709} C_VEL
LIN {X 0,Y 117.503,Z 381.242,A -85,B 0,C 180,E1 -27501.044,E2 -27501.044} C_VEL
LIN {X 0,Y 125.245,Z 376.271,A -85,B 0,C 180,E1 -27504.461,E2 -27504.461} C_VEL
LIN {X 0,Y 134.868,Z 369.189,A -85,B 0,C 180,E1 -27507.871,E2 -27507.871} C_VEL
LIN {X 0,Y 143.614,Z 361.587,A -85,B 0,C 180,E1 -27510.561,E2 -27510.561} C_VEL
LIN {X 0,Y 152.173,Z 353.016,A -85,B 0,C 180,E1 -27512.761,E2 -27512.761} C_VEL
LIN {X 0,Y 161.297,Z 342.363,A -85,B 0,C 180,E1 -27514.712,E2 -27514.712} C_VEL
LIN {X 0,Y 166.653,Z 335.096,A -85,B 0,C 180,E1 -27515.802,E2 -27515.802} C_VEL
LIN {X 0,Y 169.527,Z 330.512,A -85,B 0,C 180,E1 -27516.571,E2 -27516.571} C_VEL
LIN {X 0,Y 173.451,Z 322.848,A -85,B 0,C 180,E1 -27518.253,E2 -27518.253} C_VEL
LIN {X 0,Y 177.089,Z 314.957,A -85,B 0,C 180,E1 -27519.799,E2 -27519.799} C_VEL
LIN {X 0,Y 179.427,Z 309.842,A -85,B 0,C 180,E1 -27520.367,E2 -27520.367} C_VEL
LIN {X 0,Y 185.227,Z 295.858,A -85,B 0,C 180,E1 -27521.128,E2 -27521.128} C_VEL
LIN {X 0,Y 189.564,Z 281.991,A -85,B 0,C 180,E1 -27521.626,E2 -27521.626} C_VEL
LIN {X 0,Y 192.562,Z 267.873,A -85,B 0,C 180,E1 -27522.051,E2 -27522.051} C_VEL
LIN {X 0,Y 192.822,Z 265.827,A -85,B 0,C 180,E1 -27522.188,E2 -27522.188} C_VEL
LIN {X 0,Y 191.951,Z 262.175,A -85,B 0,C 180,E1 -27524.872,E2 -27524.872} C_VEL
LIN {X 0,Y 191.469,Z 260.525,A -85,B 0,C 180,E1 -27526.731,E2 -27526.731} C_VEL
LIN {X 0,Y 190.873,Z 257.786,A -85,B 0,C 180,E1 -27532.504,E2 -27532.504} C_VEL
LIN {X 0,Y 190.958,Z 257.882,A -85,B 0,C 180,E1 -27533.874,E2 -27533.874} C_VEL
LIN {X 0,Y 191.777,Z 261.047,A -85,B 0,C 180,E1 -27538.812,E2 -27538.812} C_VEL
LIN {X 0,Y 192.608,Z 263.857,A -85,B 0,C 180,E1 -27541.431,E2 -27541.431} C_VEL
LIN {X 0,Y 192.944,Z 264.909,A -85,B 0,C 180,E1 -27542.279,E2 -27542.279} C_VEL
LIN {X 0,Y 189.853,Z 279.76,A -85,B 0,C 180,E1 -27542.735,E2 -27542.735} C_VEL
LIN {X 0,Y 185.704,Z 293.222,A -85,B 0,C 180,E1 -27543.258,E2 -27543.258} C_VEL
LIN {X 0,Y 180.704,Z 305.752,A -85,B 0,C 180,E1 -27544.056,E2 -27544.056} C_VEL
LIN {X 0,Y 174.626,Z 317.841,A -85,B 0,C 180,E1 -27545.035,E2 -27545.035} C_VEL
LIN {X 0,Y 167.07,Z 330.066,A -85,B 0,C 180,E1 -27546.349,E2 -27546.349} C_VEL
LIN {X 0,Y 158.595,Z 341.362,A -85,B 0,C 180,E1 -27547.943,E2 -27547.943} C_VEL
LIN {X 0,Y 149.802,Z 351.204,A -85,B 0,C 180,E1 -27549.843,E2 -27549.843} C_VEL
LIN {X 0,Y 140.256,Z 360.281,A -85,B 0,C 180,E1 -27552.264,E2 -27552.264} C_VEL
LIN {X 0,Y 130.972,Z 367.733,A -85,B 0,C 180,E1 -27554.993,E2 -27554.993} C_VEL
LIN {X 0,Y 122.04,Z 373.85,A -85,B 0,C 180,E1 -27558.146,E2 -27558.146} C_VEL
LIN {X 0,Y 113.555,Z 378.826,A -85,B 0,C 180,E1 -27561.807,E2 -27561.807} C_VEL
LIN {X 0,Y 105.6,Z 382.788,A -85,B 0,C 180,E1 -27566.031,E2 -27566.031} C_VEL
LIN {X 0,Y 98.278,Z 385.795,A -85,B 0,C 180,E1 -27570.881,E2 -27570.881} C_VEL
LIN {X 0,Y 89.832,Z 388.416,A -85,B 0,C 180,E1 -27578.514,E2 -27578.514} C_VEL
LIN {X 0,Y 83.196,Z 389.528,A -85,B 0,C 180,E1 -27587.475,E2 -27587.475} C_VEL
LIN {X 0,Y 78.671,Z 389.198,A -85,B 0,C 180,E1 -27597.58,E2 -27597.58} C_VEL
LIN {X 0,Y 76.533,Z 387.436,A -85,B 0,C 180,E1 -27608.442,E2 -27608.442} C_VEL
LIN {X 0,Y 76.349,Z 384.255,A -85,B 0,C 180,E1 -27619.384,E2 -27619.384} C_VEL
LIN {X 0,Y 77.436,Z 381.353,A -85,B 0,C 180,E1 -27626.383,E2 -27626.383} C_VEL
LIN {X 0,Y 79.815,Z 376.613,A -85,B 0,C 180,E1 -27635.044,E2 -27635.044} C_VEL
LIN {X 0,Y 83.627,Z 370.394,A -85,B 0,C 180,E1 -27643.355,E2 -27643.355} C_VEL
LIN {X 0,Y 88.885,Z 362.63,A -85,B 0,C 180,E1 -27650.836,E2 -27650.836} C_VEL
LIN {X 0,Y 94.324,Z 354.537,A -85,B 0,C 180,E1 -27656.548,E2 -27656.548} C_VEL
LIN {X 0,Y 100.348,Z 344.81,A -85,B 0,C 180,E1 -27661.68,E2 -27661.68} C_VEL
LIN {X 0,Y 106.009,Z 335.058,A -85,B 0,C 180,E1 -27665.45,E2 -27665.45} C_VEL
LIN {X 0,Y 111.404,Z 324.584,A -85,B 0,C 180,E1 -27668.526,E2 -27668.526} C_VEL
LIN {X 0,Y 117.151,Z 311.746,A -85,B 0,C 180,E1 -27671.285,E2 -27671.285} C_VEL
LIN {X 0,Y 121.739,Z 299.251,A -85,B 0,C 180,E1 -27673.272,E2 -27673.272} C_VEL
LIN {X 0,Y 125.314,Z 286.748,A -85,B 0,C 180,E1 -27674.786,E2 -27674.786} C_VEL
LIN {X 0,Y 128.19,Z 273.31,A -85,B 0,C 180,E1 -27675.945,E2 -27675.945} C_VEL
LIN {X 0,Y 130.374,Z 258.405,A -85,B 0,C 180,E1 -27676.691,E2 -27676.691} C_VEL
LIN {X 0,Y 134.223,Z 218.171,A -85,B 0,C 180,E1 -27678.152,E2 -27678.152} C_VEL
LIN {X 0,Y 130.223,Z 208.824,A -85,B 0,C 180,E1 -27682.022,E2 -27682.022} C_VEL
LIN {X 0,Y 127.134,Z 202.583,A -85,B 0,C 180,E1 -27685.437,E2 -27685.437} C_VEL
LIN {X 0,Y 124.379,Z 197.49,A -85,B 0,C 180,E1 -27688.969,E2 -27688.969} C_VEL
LIN {X 0,Y 122.757,Z 194.742,A -85,B 0,C 180,E1 -27691.344,E2 -27691.344} C_VEL
LIN {X 0,Y 120.948,Z 191.628,A -85,B 0,C 180,E1 -27694.452,E2 -27694.452} C_VEL
LIN {X 0,Y 118.683,Z 187.765,A -85,B 0,C 180,E1 -27699.539,E2 -27699.539} C_VEL
LIN {X 0,Y 116.709,Z 184.243,A -85,B 0,C 180,E1 -27708.245,E2 -27708.245} C_VEL
LIN {X 0,Y 116.665,Z 183.052,A -85,B 0,C 180,E1 -27710.574,E2 -27710.574} C_VEL
LIN {X 0,Y 116.871,Z 183.159,A -85,B 0,C 180,E1 -27715.595,E2 -27715.595} C_VEL
LIN {X 0,Y 117.781,Z 186.346,A -85,B 0,C 180,E1 -27721.3,E2 -27721.3} C_VEL
LIN {X 0,Y 119.047,Z 187.972,A -85,B 0,C 180,E1 -27724.942,E2 -27724.942} C_VEL
LIN {X 0,Y 121.242,Z 191.77,A -85,B 0,C 180,E1 -27729.646,E2 -27729.646} C_VEL
LIN {X 0,Y 123.736,Z 196.282,A -85,B 0,C 180,E1 -27733.731,E2 -27733.731} C_VEL
LIN {X 0,Y 126.874,Z 202,A -85,B 0,C 180,E1 -27737.879,E2 -27737.879} C_VEL
LIN {X 0,Y 130.325,Z 209.176,A -85,B 0,C 180,E1 -27741.733,E2 -27741.733} C_VEL
LIN {X 0,Y 131.99,Z 213.091,A -85,B 0,C 180,E1 -27743.418,E2 -27743.418} C_VEL
LIN {X 0,Y 134.168,Z 220.794,A -85,B 0,C 180,E1 -27745.7,E2 -27745.7} C_VEL
LIN {X 0,Y 129.52,Z 268.671,A -85,B 0,C 180,E1 -27747.518,E2 -27747.518} C_VEL
LIN {X 0,Y 126.883,Z 283.401,A -85,B 0,C 180,E1 -27748.451,E2 -27748.451} C_VEL
LIN {X 0,Y 123.429,Z 296.878,A -85,B 0,C 180,E1 -27749.745,E2 -27749.745} C_VEL
LIN {X 0,Y 118.608,Z 310.923,A -85,B 0,C 180,E1 -27751.604,E2 -27751.604} C_VEL
LIN {X 0,Y 113.23,Z 323.642,A -85,B 0,C 180,E1 -27753.973,E2 -27753.973} C_VEL
LIN {X 0,Y 108.27,Z 333.816,A -85,B 0,C 180,E1 -27756.564,E2 -27756.564} C_VEL
LIN {X 0,Y 104.015,Z 341.583,A -85,B 0,C 180,E1 -27759.021,E2 -27759.021} C_VEL
LIN {X 0,Y 98.317,Z 351.05,A -85,B 0,C 180,E1 -27762.895,E2 -27762.895} C_VEL
LIN {X 0,Y 92.178,Z 360.525,A -85,B 0,C 180,E1 -27768.162,E2 -27768.162} C_VEL
LIN {X 0,Y 87.198,Z 367.94,A -85,B 0,C 180,E1 -27773.728,E2 -27773.728} C_VEL
LIN {X 0,Y 83.309,Z 373.873,A -85,B 0,C 180,E1 -27779.599,E2 -27779.599} C_VEL
LIN {X 0,Y 79.988,Z 379.434,A -85,B 0,C 180,E1 -27786.718,E2 -27786.718} C_VEL
LIN {X 0,Y 77.381,Z 385.237,A -85,B 0,C 180,E1 -27796.884,E2 -27796.884} C_VEL
LIN {X 0,Y 76.74,Z 388.512,A -85,B 0,C 180,E1 -27804.753,E2 -27804.753} C_VEL
LIN {X 0,Y 76.797,Z 390.199,A -85,B 0,C 180,E1 -27810.007,E2 -27810.007} C_VEL
LIN {X 0,Y 76.786,Z 391.5,A -85,B 0,C 180,E1 -27815.259,E2 -27815.259} C_VEL
LIN {X 0,Y 77.973,Z 393.082,A -85,B 0,C 180,E1 -27825.696,E2 -27825.696} C_VEL
LIN {X 0,Y 81.321,Z 393.368,A -85,B 0,C 180,E1 -27835.609,E2 -27835.609} C_VEL
LIN {X 0,Y 86.952,Z 392.384,A -85,B 0,C 180,E1 -27844.465,E2 -27844.465} C_VEL
LIN {X 0,Y 94.341,Z 390.109,A -85,B 0,C 180,E1 -27852.11,E2 -27852.11} C_VEL
LIN {X 0,Y 103.166,Z 386.486,A -85,B 0,C 180,E1 -27858.543,E2 -27858.543} C_VEL
LIN {X 0,Y 113.158,Z 381.411,A -85,B 0,C 180,E1 -27863.851,E2 -27863.851} C_VEL
LIN {X 0,Y 121.26,Z 376.538,A -85,B 0,C 180,E1 -27867.19,E2 -27867.19} C_VEL
LIN {X 0,Y 131.242,Z 369.563,A -85,B 0,C 180,E1 -27870.489,E2 -27870.489} C_VEL
LIN {X 0,Y 139.842,Z 362.47,A -85,B 0,C 180,E1 -27872.967,E2 -27872.967} C_VEL
LIN {X 0,Y 149.08,Z 353.647,A -85,B 0,C 180,E1 -27875.169,E2 -27875.169} C_VEL
LIN {X 0,Y 158.42,Z 343.171,A -85,B 0,C 180,E1 -27877.012,E2 -27877.012} C_VEL
LIN {X 0,Y 166.253,Z 332.677,A -85,B 0,C 180,E1 -27878.444,E2 -27878.444} C_VEL
LIN {X 0,Y 173.48,Z 321.236,A -85,B 0,C 180,E1 -27879.535,E2 -27879.535} C_VEL
LIN {X 0,Y 179.427,Z 309.842,A -85,B 0,C 180,E1 -27880.367,E2 -27880.367} C_VEL
LIN {X 0,Y 182.291,Z 302.889,A -85,B 0,C 180,E1 -27881.087,E2 -27881.087} C_VEL
LIN {X 0,Y 186.508,Z 289.048,A -85,B 0,C 180,E1 -27883.072,E2 -27883.072} C_VEL
LIN {X 0,Y 188.402,Z 281.735,A -85,B 0,C 180,E1 -27883.748,E2 -27883.748} C_VEL
LIN {X 0,Y 190.867,Z 270.656,A -85,B 0,C 180,E1 -27884.098,E2 -27884.098} C_VEL
LIN {X 0,Y 190.519,Z 268.486,A -85,B 0,C 180,E1 -27885.848,E2 -27885.848} C_VEL
LIN {X 0,Y 190.265,Z 267.373,A -85,B 0,C 180,E1 -27887.189,E2 -27887.189} C_VEL
LIN {X 0,Y 189.872,Z 264.822,A -85,B 0,C 180,E1 -27892.55,E2 -27892.55} C_VEL
LIN {X 0,Y 189.94,Z 265.129,A -85,B 0,C 180,E1 -27894.061,E2 -27894.061} C_VEL
LIN {X 0,Y 190.453,Z 267.758,A -85,B 0,C 180,E1 -27898.239,E2 -27898.239} C_VEL
LIN {X 0,Y 190.917,Z 269.785,A -85,B 0,C 180,E1 -27900.294,E2 -27900.294} C_VEL
LIN {X 0,Y 187.437,Z 284.265,A -85,B 0,C 180,E1 -27900.753,E2 -27900.753} C_VEL
LIN {X 0,Y 183.247,Z 296.621,A -85,B 0,C 180,E1 -27901.271,E2 -27901.271} C_VEL
LIN {X 0,Y 177.884,Z 309.027,A -85,B 0,C 180,E1 -27902.044,E2 -27902.044} C_VEL
LIN {X 0,Y 171.548,Z 320.78,A -85,B 0,C 180,E1 -27902.979,E2 -27902.979} C_VEL
LIN {X 0,Y 163.854,Z 332.519,A -85,B 0,C 180,E1 -27904.218,E2 -27904.218} C_VEL
LIN {X 0,Y 155.389,Z 343.204,A -85,B 0,C 180,E1 -27905.683,E2 -27905.683} C_VEL
LIN {X 0,Y 145.4,Z 353.707,A -85,B 0,C 180,E1 -27907.717,E2 -27907.717} C_VEL
LIN {X 0,Y 135.612,Z 362.335,A -85,B 0,C 180,E1 -27910.025,E2 -27910.025} C_VEL
LIN {X 0,Y 125.258,Z 370.011,A -85,B 0,C 180,E1 -27912.958,E2 -27912.958} C_VEL
LIN {X 0,Y 113.896,Z 376.991,A -85,B 0,C 180,E1 -27916.958,E2 -27916.958} C_VEL
LIN {X 0,Y 105.265,Z 381.372,A -85,B 0,C 180,E1 -27920.805,E2 -27920.805} C_VEL
LIN {X 0,Y 94.606,Z 385.711,A -85,B 0,C 180,E1 -27926.932,E2 -27926.932} C_VEL
LIN {X 0,Y 85.313,Z 388.472,A -85,B 0,C 180,E1 -27934.523,E2 -27934.523} C_VEL
LIN {X 0,Y 77.783,Z 389.709,A -85,B 0,C 180,E1 -27943.701,E2 -27943.701} C_VEL
LIN {X 0,Y 72.446,Z 389.482,A -85,B 0,C 180,E1 -27954.395,E2 -27954.395} C_VEL
LIN {X 0,Y 69.686,Z 387.82,A -85,B 0,C 180,E1 -27966.2,E2 -27966.2} C_VEL
LIN {X 0,Y 69.124,Z 386.46,A -85,B 0,C 180,E1 -27972.232,E2 -27972.232} C_VEL
LIN {X 0,Y 69.855,Z 382.642,A -85,B 0,C 180,E1 -27984.218,E2 -27984.218} C_VEL
LIN {X 0,Y 71.783,Z 378.76,A -85,B 0,C 180,E1 -27992.798,E2 -27992.798} C_VEL
LIN {X 0,Y 74.717,Z 373.983,A -85,B 0,C 180,E1 -28000.835,E2 -28000.835} C_VEL
LIN {X 0,Y 79.696,Z 367.038,A -85,B 0,C 180,E1 -28009.303,E2 -28009.303} C_VEL
LIN {X 0,Y 86.028,Z 358.424,A -85,B 0,C 180,E1 -28016.692,E2 -28016.692} C_VEL
LIN {X 0,Y 92.279,Z 349.441,A -85,B 0,C 180,E1 -28022.209,E2 -28022.209} C_VEL
LIN {X 0,Y 97.763,Z 340.584,A -85,B 0,C 180,E1 -28026.368,E2 -28026.368} C_VEL
LIN {X 0,Y 104.099,Z 329.9,A -85,B 0,C 180,E1 -28029.887,E2 -28029.887} C_VEL
LIN {X 0,Y 109.894,Z 318.306,A -85,B 0,C 180,E1 -28032.797,E2 -28032.797} C_VEL
LIN {X 0,Y 115.273,Z 305.565,A -85,B 0,C 180,E1 -28035.127,E2 -28035.127} C_VEL
LIN {X 0,Y 119.688,Z 292.428,A -85,B 0,C 180,E1 -28036.906,E2 -28036.906} C_VEL
LIN {X 0,Y 123.391,Z 278.044,A -85,B 0,C 180,E1 -28038.254,E2 -28038.254} C_VEL
LIN {X 0,Y 125.428,Z 266.554,A -85,B 0,C 180,E1 -28039,E2 -28039} C_VEL
LIN {X 0,Y 128.439,Z 239.361,A -85,B 0,C 180,E1 -28039.994,E2 -28039.994} C_VEL
LIN {X 0,Y 130.194,Z 221.045,A -85,B 0,C 180,E1 -28040.682,E2 -28040.682} C_VEL
LIN {X 0,Y 126.998,Z 213.175,A -85,B 0,C 180,E1 -28044.206,E2 -28044.206} C_VEL
LIN {X 0,Y 124.257,Z 207.263,A -85,B 0,C 180,E1 -28047.652,E2 -28047.652} C_VEL
LIN {X 0,Y 121.373,Z 201.683,A -85,B 0,C 180,E1 -28051.942,E2 -28051.942} C_VEL
LIN {X 0,Y 119.443,Z 198.264,A -85,B 0,C 180,E1 -28055.465,E2 -28055.465} C_VEL
LIN {X 0,Y 117.504,Z 194.625,A -85,B 0,C 180,E1 -28060.238,E2 -28060.238} C_VEL
LIN {X 0,Y 115.772,Z 191.166,A -85,B 0,C 180,E1 -28068.834,E2 -28068.834} C_VEL
LIN {X 0,Y 115.765,Z 190.022,A -85,B 0,C 180,E1 -28071.479,E2 -28071.479} C_VEL
LIN {X 0,Y 115.921,Z 190.215,A -85,B 0,C 180,E1 -28075.07,E2 -28075.07} C_VEL
LIN {X 0,Y 116.756,Z 193.315,A -85,B 0,C 180,E1 -28080.878,E2 -28080.878} C_VEL
LIN {X 0,Y 117.776,Z 194.793,A -85,B 0,C 180,E1 -28084.083,E2 -28084.083} C_VEL
LIN {X 0,Y 120.107,Z 199.212,A -85,B 0,C 180,E1 -28089.414,E2 -28089.414} C_VEL
LIN {X 0,Y 122.143,Z 203.153,A -85,B 0,C 180,E1 -28092.92,E2 -28092.92} C_VEL
LIN {X 0,Y 125.062,Z 208.984,A -85,B 0,C 180,E1 -28097.054,E2 -28097.054} C_VEL
LIN {X 0,Y 127.956,Z 215.529,A -85,B 0,C 180,E1 -28100.546,E2 -28100.546} C_VEL
LIN {X 0,Y 129.098,Z 218.808,A -85,B 0,C 180,E1 -28101.858,E2 -28101.858} C_VEL
LIN {X 0,Y 130.199,Z 223.072,A -85,B 0,C 180,E1 -28103.174,E2 -28103.174} C_VEL
LIN {X 0,Y 125.556,Z 268.845,A -85,B 0,C 180,E1 -28104.885,E2 -28104.885} C_VEL
LIN {X 0,Y 122.893,Z 283.132,A -85,B 0,C 180,E1 -28105.76,E2 -28105.76} C_VEL
LIN {X 0,Y 119.314,Z 296.633,A -85,B 0,C 180,E1 -28107.023,E2 -28107.023} C_VEL
LIN {X 0,Y 114.31,Z 310.689,A -85,B 0,C 180,E1 -28108.834,E2 -28108.834} C_VEL
LIN {X 0,Y 108.597,Z 323.619,A -85,B 0,C 180,E1 -28111.193,E2 -28111.193} C_VEL
LIN {X 0,Y 103.502,Z 333.595,A -85,B 0,C 180,E1 -28113.727,E2 -28113.727} C_VEL
LIN {X 0,Y 99.017,Z 341.363,A -85,B 0,C 180,E1 -28116.171,E2 -28116.171} C_VEL
LIN {X 0,Y 92.404,Z 351.676,A -85,B 0,C 180,E1 -28120.495,E2 -28120.495} C_VEL
LIN {X 0,Y 85.936,Z 361.005,A -85,B 0,C 180,E1 -28125.971,E2 -28125.971} C_VEL
LIN {X 0,Y 80.301,Z 368.747,A -85,B 0,C 180,E1 -28132.228,E2 -28132.228} C_VEL
LIN {X 0,Y 75.84,Z 375.197,A -85,B 0,C 180,E1 -28139.367,E2 -28139.367} C_VEL
LIN {X 0,Y 72.441,Z 380.455,A -85,B 0,C 180,E1 -28147.175,E2 -28147.175} C_VEL
LIN {X 0,Y 70.461,Z 384.721,A -85,B 0,C 180,E1 -28155.569,E2 -28155.569} C_VEL
LIN {X 0,Y 69.655,Z 388.086,A -85,B 0,C 180,E1 -28164.217,E2 -28164.217} C_VEL
LIN {X 0,Y 69.718,Z 389.818,A -85,B 0,C 180,E1 -28170.008,E2 -28170.008} C_VEL
LIN {X 0,Y 69.727,Z 391.161,A -85,B 0,C 180,E1 -28175.793,E2 -28175.793} C_VEL
LIN {X 0,Y 71.141,Z 392.823,A -85,B 0,C 180,E1 -28187.248,E2 -28187.248} C_VEL
LIN {X 0,Y 74.958,Z 393.192,A -85,B 0,C 180,E1 -28197.965,E2 -28197.965} C_VEL
LIN {X 0,Y 81.171,Z 392.29,A -85,B 0,C 180,E1 -28207.315,E2 -28207.315} C_VEL
LIN {X 0,Y 89.18,Z 390.099,A -85,B 0,C 180,E1 -28215.184,E2 -28215.184} C_VEL
LIN {X 0,Y 98.599,Z 386.563,A -85,B 0,C 180,E1 -28221.643,E2 -28221.643} C_VEL
LIN {X 0,Y 109.107,Z 381.58,A -85,B 0,C 180,E1 -28226.873,E2 -28226.873} C_VEL
LIN {X 0,Y 120.466,Z 375.001,A -85,B 0,C 180,E1 -28231.066,E2 -28231.066} C_VEL
LIN {X 0,Y 130.914,Z 367.729,A -85,B 0,C 180,E1 -28234.063,E2 -28234.063} C_VEL
LIN {X 0,Y 139.845,Z 360.299,A -85,B 0,C 180,E1 -28236.342,E2 -28236.342} C_VEL
LIN {X 0,Y 149.426,Z 351.103,A -85,B 0,C 180,E1 -28238.275,E2 -28238.275} C_VEL
LIN {X 0,Y 158.998,Z 340.167,A -85,B 0,C 180,E1 -28239.942,E2 -28239.942} C_VEL
LIN {X 0,Y 166.241,Z 330.266,A -85,B 0,C 180,E1 -28241.081,E2 -28241.081} C_VEL
LIN {X 0,Y 173.617,Z 318.347,A -85,B 0,C 180,E1 -28242.051,E2 -28242.051} C_VEL
LIN {X 0,Y 180.19,Z 305.126,A -85,B 0,C 180,E1 -28242.868,E2 -28242.868} C_VEL
LIN {X 0,Y 185.404,Z 291.648,A -85,B 0,C 180,E1 -28243.459,E2 -28243.459} C_VEL
LIN {X 0,Y 188.402,Z 281.735,A -85,B 0,C 180,E1 -28243.748,E2 -28243.748} C_VEL
LIN {X 0,Y 188.92,Z 279.273,A -85,B 0,C 180,E1 -28244.117,E2 -28244.117} C_VEL
LIN {X 0,Y 189.145,Z 277.007,A -85,B 0,C 180,E1 -28244.94,E2 -28244.94} C_VEL
LIN {X 0,Y 189.075,Z 275.428,A -85,B 0,C 180,E1 -28246.051,E2 -28246.051} C_VEL
LIN {X 0,Y 188.52,Z 273.208,A -85,B 0,C 180,E1 -28249.685,E2 -28249.685} C_VEL
LIN {X 0,Y 188.561,Z 271.849,A -85,B 0,C 180,E1 -28252.498,E2 -28252.498} C_VEL
LIN {X 0,Y 188.602,Z 272.217,A -85,B 0,C 180,E1 -28254.111,E2 -28254.111} C_VEL
LIN {X 0,Y 188.858,Z 274.496,A -85,B 0,C 180,E1 -28257.738,E2 -28257.738} C_VEL
LIN {X 0,Y 188.917,Z 275.054,A -85,B 0,C 180,E1 -28258.313,E2 -28258.313} C_VEL
LIN {X 0,Y 185.011,Z 289.012,A -85,B 0,C 180,E1 -28258.751,E2 -28258.751} C_VEL
LIN {X 0,Y 180.113,Z 301.912,A -85,B 0,C 180,E1 -28259.334,E2 -28259.334} C_VEL
LIN {X 0,Y 174.019,Z 314.497,A -85,B 0,C 180,E1 -28260.136,E2 -28260.136} C_VEL
LIN {X 0,Y 166.954,Z 326.26,A -85,B 0,C 180,E1 -28261.091,E2 -28261.091} C_VEL
LIN {X 0,Y 158.149,Z 338.314,A -85,B 0,C 180,E1 -28262.428,E2 -28262.428} C_VEL
LIN {X 0,Y 149.684,Z 347.903,A -85,B 0,C 180,E1 -28263.808,E2 -28263.808} C_VEL
LIN {X 0,Y 139.635,Z 357.514,A -85,B 0,C 180,E1 -28265.768,E2 -28265.768} C_VEL
LIN {X 0,Y 129.541,Z 365.587,A -85,B 0,C 180,E1 -28268.034,E2 -28268.034} C_VEL
LIN {X 0,Y 118.215,Z 373.12,A -85,B 0,C 180,E1 -28271.181,E2 -28271.181} C_VEL
LIN {X 0,Y 106.534,Z 379.446,A -85,B 0,C 180,E1 -28275.287,E2 -28275.287} C_VEL
LIN {X 0,Y 97.001,Z 383.611,A -85,B 0,C 180,E1 -28279.613,E2 -28279.613} C_VEL
LIN {X 0,Y 86.148,Z 387.253,A -85,B 0,C 180,E1 -28286.17,E2 -28286.17} C_VEL
LIN {X 0,Y 76.751,Z 389.368,A -85,B 0,C 180,E1 -28294.488,E2 -28294.488} C_VEL
LIN {X 0,Y 69.29,Z 390.006,A -85,B 0,C 180,E1 -28304.753,E2 -28304.753} C_VEL
LIN {X 0,Y 64.312,Z 389.167,A -85,B 0,C 180,E1 -28316.869,E2 -28316.869} C_VEL
LIN {X 0,Y 62.922,Z 388.206,A -85,B 0,C 180,E1 -28323.453,E2 -28323.453} C_VEL
LIN {X 0,Y 62.133,Z 386.893,A -85,B 0,C 180,E1 -28330.154,E2 -28330.154} C_VEL
LIN {X 0,Y 62.576,Z 383.179,A -85,B 0,C 180,E1 -28343.542,E2 -28343.542} C_VEL
LIN {X 0,Y 64.59,Z 379.4,A -85,B 0,C 180,E1 -28353.11,E2 -28353.11} C_VEL
LIN {X 0,Y 67.7,Z 374.722,A -85,B 0,C 180,E1 -28361.974,E2 -28361.974} C_VEL
LIN {X 0,Y 72.955,Z 367.925,A -85,B 0,C 180,E1 -28371.168,E2 -28371.168} C_VEL
LIN {X 0,Y 78.68,Z 360.797,A -85,B 0,C 180,E1 -28377.958,E2 -28377.958} C_VEL
LIN {X 0,Y 85.213,Z 352.13,A -85,B 0,C 180,E1 -28383.945,E2 -28383.945} C_VEL
LIN {X 0,Y 92.134,Z 341.973,A -85,B 0,C 180,E1 -28388.991,E2 -28388.991} C_VEL
LIN {X 0,Y 98.681,Z 331.552,A -85,B 0,C 180,E1 -28392.569,E2 -28392.569} C_VEL
LIN {X 0,Y 104.794,Z 320.243,A -85,B 0,C 180,E1 -28395.436,E2 -28395.436} C_VEL
LIN {X 0,Y 110.381,Z 307.913,A -85,B 0,C 180,E1 -28397.738,E2 -28397.738} C_VEL
LIN {X 0,Y 115.323,Z 294.241,A -85,B 0,C 180,E1 -28399.613,E2 -28399.613} C_VEL
LIN {X 0,Y 119.068,Z 280.579,A -85,B 0,C 180,E1 -28400.952,E2 -28400.952} C_VEL
LIN {X 0,Y 121.536,Z 268.352,A -85,B 0,C 180,E1 -28401.731,E2 -28401.731} C_VEL
LIN {X 0,Y 123.823,Z 249.881,A -85,B 0,C 180,E1 -28402.436,E2 -28402.436} C_VEL
LIN {X 0,Y 126.434,Z 223.913,A -85,B 0,C 180,E1 -28403.37,E2 -28403.37} C_VEL
LIN {X 0,Y 123.422,Z 216.15,A -85,B 0,C 180,E1 -28407.25,E2 -28407.25} C_VEL
LIN {X 0,Y 120.487,Z 209.849,A -85,B 0,C 180,E1 -28411.674,E2 -28411.674} C_VEL
LIN {X 0,Y 118.091,Z 205.031,A -85,B 0,C 180,E1 -28416.268,E2 -28416.268} C_VEL
LIN {X 0,Y 116.159,Z 201.292,A -85,B 0,C 180,E1 -28421.515,E2 -28421.515} C_VEL
LIN {X 0,Y 114.844,Z 197.585,A -85,B 0,C 180,E1 -28430.547,E2 -28430.547} C_VEL
LIN {X 0,Y 114.875,Z 197.126,A -85,B 0,C 180,E1 -28431.413,E2 -28431.413} C_VEL
LIN {X 0,Y 114.988,Z 197.394,A -85,B 0,C 180,E1 -28434.784,E2 -28434.784} C_VEL
LIN {X 0,Y 115.847,Z 200.474,A -85,B 0,C 180,E1 -28440.885,E2 -28440.885} C_VEL
LIN {X 0,Y 116.484,Z 201.47,A -85,B 0,C 180,E1 -28443.04,E2 -28443.04} C_VEL
LIN {X 0,Y 118.555,Z 205.785,A -85,B 0,C 180,E1 -28448.319,E2 -28448.319} C_VEL
LIN {X 0,Y 120.435,Z 209.735,A -85,B 0,C 180,E1 -28451.856,E2 -28451.856} C_VEL
LIN {X 0,Y 123.282,Z 215.915,A -85,B 0,C 180,E1 -28456.202,E2 -28456.202} C_VEL
LIN {X 0,Y 125.702,Z 222.128,A -85,B 0,C 180,E1 -28459.399,E2 -28459.399} C_VEL
LIN {X 0,Y 126.49,Z 225.367,A -85,B 0,C 180,E1 -28460.489,E2 -28460.489} C_VEL
LIN {X 0,Y 121.864,Z 268.987,A -85,B 0,C 180,E1 -28462.073,E2 -28462.073} C_VEL
LIN {X 0,Y 119.009,Z 283.637,A -85,B 0,C 180,E1 -28462.958,E2 -28462.958} C_VEL
LIN {X 0,Y 115.099,Z 297.515,A -85,B 0,C 180,E1 -28464.217,E2 -28464.217} C_VEL
LIN {X 0,Y 110.3,Z 310.455,A -85,B 0,C 180,E1 -28465.855,E2 -28465.855} C_VEL
LIN {X 0,Y 104.272,Z 323.542,A -85,B 0,C 180,E1 -28468.165,E2 -28468.165} C_VEL
LIN {X 0,Y 98.997,Z 333.4,A -85,B 0,C 180,E1 -28470.63,E2 -28470.63} C_VEL
LIN {X 0,Y 94.288,Z 341.143,A -85,B 0,C 180,E1 -28473.025,E2 -28473.025} C_VEL
LIN {X 0,Y 87.914,Z 350.618,A -85,B 0,C 180,E1 -28476.937,E2 -28476.937} C_VEL
LIN {X 0,Y 80.922,Z 360.103,A -85,B 0,C 180,E1 -28482.431,E2 -28482.431} C_VEL
LIN {X 0,Y 74.118,Z 368.735,A -85,B 0,C 180,E1 -28489.636,E2 -28489.636} C_VEL
LIN {X 0,Y 69.734,Z 374.484,A -85,B 0,C 180,E1 -28496.347,E2 -28496.347} C_VEL
LIN {X 0,Y 65.9,Z 379.84,A -85,B 0,C 180,E1 -28504.759,E2 -28504.759} C_VEL
LIN {X 0,Y 63.105,Z 385.461,A -85,B 0,C 180,E1 -28517.139,E2 -28517.139} C_VEL
LIN {X 0,Y 62.584,Z 387.645,A -85,B 0,C 180,E1 -28523.562,E2 -28523.562} C_VEL
LIN {X 0,Y 62.628,Z 389.433,A -85,B 0,C 180,E1 -28530.009,E2 -28530.009} C_VEL
LIN {X 0,Y 62.649,Z 390.82,A -85,B 0,C 180,E1 -28536.45,E2 -28536.45} C_VEL
LIN {X 0,Y 64.377,Z 392.565,A -85,B 0,C 180,E1 -28549.127,E2 -28549.127} C_VEL
LIN {X 0,Y 68.749,Z 393.016,A -85,B 0,C 180,E1 -28560.749,E2 -28560.749} C_VEL
LIN {X 0,Y 75.623,Z 392.196,A -85,B 0,C 180,E1 -28570.592,E2 -28570.592} C_VEL
LIN {X 0,Y 84.296,Z 390.088,A -85,B 0,C 180,E1 -28578.631,E2 -28578.631} C_VEL
LIN {X 0,Y 94.336,Z 386.641,A -85,B 0,C 180,E1 -28585.044,E2 -28585.044} C_VEL
LIN {X 0,Y 105.385,Z 381.762,A -85,B 0,C 180,E1 -28590.117,E2 -28590.117} C_VEL
LIN {X 0,Y 117.202,Z 375.297,A -85,B 0,C 180,E1 -28594.099,E2 -28594.099} C_VEL
LIN {X 0,Y 127.969,Z 368.141,A -85,B 0,C 180,E1 -28596.922,E2 -28596.922} C_VEL
LIN {X 0,Y 137.326,Z 360.704,A -85,B 0,C 180,E1 -28599.076,E2 -28599.076} C_VEL
LIN {X 0,Y 146.956,Z 351.791,A -85,B 0,C 180,E1 -28600.836,E2 -28600.836} C_VEL
LIN {X 0,Y 156.726,Z 341.034,A -85,B 0,C 180,E1 -28602.356,E2 -28602.356} C_VEL
LIN {X 0,Y 164.922,Z 330.179,A -85,B 0,C 180,E1 -28603.511,E2 -28603.511} C_VEL
LIN {X 0,Y 172.418,Z 318.28,A -85,B 0,C 180,E1 -28604.374,E2 -28604.374} C_VEL
LIN {X 0,Y 179.089,Z 305.108,A -85,B 0,C 180,E1 -28605.108,E2 -28605.108} C_VEL
LIN {X 0,Y 184.382,Z 291.661,A -85,B 0,C 180,E1 -28605.633,E2 -28605.633} C_VEL
LIN {X 0,Y 188.522,Z 277.335,A -85,B 0,C 180,E1 -28606.042,E2 -28606.042} C_VEL
LIN {X 0,Y 188.952,Z 275.413,A -85,B 0,C 180,E1 -28606.143,E2 -28606.143} C_VEL
LIN {X 0,Y 188.716,Z 274.041,A -85,B 0,C 180,E1 -28607.901,E2 -28607.901} C_VEL
LIN {X 0,Y 188.52,Z 273.208,A -85,B 0,C 180,E1 -28609.685,E2 -28609.685} C_VEL
LIN {X 0,Y 188.34,Z 273.303,A -85,B 0,C 180,E1 -28610.864,E2 -28610.864} C_VEL
LIN {X 0,Y 187.968,Z 274.548,A -85,B 0,C 180,E1 -28612.007,E2 -28612.007} C_VEL
LIN {X 0,Y 186.979,Z 279.454,A -85,B 0,C 180,E1 -28614.998,E2 -28614.998} C_VEL
LIN {X 0,Y 186.912,Z 280.196,A -85,B 0,C 180,E1 -28615.81,E2 -28615.81} C_VEL
LIN {X 0,Y 186.938,Z 280.464,A -85,B 0,C 180,E1 -28616.288,E2 -28616.288} C_VEL
LIN {X 0,Y 182.469,Z 294.325,A -85,B 0,C 180,E1 -28616.727,E2 -28616.727} C_VEL
LIN {X 0,Y 176.774,Z 307.629,A -85,B 0,C 180,E1 -28617.369,E2 -28617.369} C_VEL
LIN {X 0,Y 170.103,Z 319.932,A -85,B 0,C 180,E1 -28618.156,E2 -28618.156} C_VEL
LIN {X 0,Y 162.551,Z 331.295,A -85,B 0,C 180,E1 -28619.099,E2 -28619.099} C_VEL
LIN {X 0,Y 153.749,Z 342.268,A -85,B 0,C 180,E1 -28620.301,E2 -28620.301} C_VEL
LIN {X 0,Y 144.152,Z 352.226,A -85,B 0,C 180,E1 -28621.769,E2 -28621.769} C_VEL
LIN {X 0,Y 133.817,Z 361.213,A -85,B 0,C 180,E1 -28623.682,E2 -28623.682} C_VEL
LIN {X 0,Y 123.647,Z 368.592,A -85,B 0,C 180,E1 -28625.87,E2 -28625.87} C_VEL
LIN {X 0,Y 113.697,Z 374.648,A -85,B 0,C 180,E1 -28628.469,E2 -28628.469} C_VEL
LIN {X 0,Y 103.563,Z 379.788,A -85,B 0,C 180,E1 -28631.733,E2 -28631.733} C_VEL
LIN {X 0,Y 91.724,Z 384.587,A -85,B 0,C 180,E1 -28636.692,E2 -28636.692} C_VEL
LIN {X 0,Y 83.088,Z 387.235,A -85,B 0,C 180,E1 -28641.48,E2 -28641.48} C_VEL
LIN {X 0,Y 72.729,Z 389.448,A -85,B 0,C 180,E1 -28649.562,E2 -28649.562} C_VEL
LIN {X 0,Y 64.195,Z 390.199,A -85,B 0,C 180,E1 -28659.959,E2 -28659.959} C_VEL
LIN {X 0,Y 58.16,Z 389.499,A -85,B 0,C 180,E1 -28672.817,E2 -28672.817} C_VEL
LIN {X 0,Y 56.1,Z 388.402,A -85,B 0,C 180,E1 -28681.221,E2 -28681.221} C_VEL
LIN {X 0,Y 54.844,Z 385.708,A -85,B 0,C 180,E1 -28695.139,E2 -28695.139} C_VEL
LIN {X 0,Y 56.221,Z 381.918,A -85,B 0,C 180,E1 -28708.377,E2 -28708.377} C_VEL
LIN {X 0,Y 59.456,Z 377.06,A -85,B 0,C 180,E1 -28720.203,E2 -28720.203} C_VEL
LIN {X 0,Y 64.568,Z 370.804,A -85,B 0,C 180,E1 -28730.707,E2 -28730.707} C_VEL
LIN {X 0,Y 71.352,Z 362.999,A -85,B 0,C 180,E1 -28739.495,E2 -28739.495} C_VEL
LIN {X 0,Y 77.696,Z 355.421,A -85,B 0,C 180,E1 -28745.409,E2 -28745.409} C_VEL
LIN {X 0,Y 84.224,Z 346.875,A -85,B 0,C 180,E1 -28750.283,E2 -28750.283} C_VEL
LIN {X 0,Y 90.742,Z 337.445,A -85,B 0,C 180,E1 -28754.182,E2 -28754.182} C_VEL
LIN {X 0,Y 97.045,Z 327.284,A -85,B 0,C 180,E1 -28757.151,E2 -28757.151} C_VEL
LIN {X 0,Y 103.544,Z 314.959,A -85,B 0,C 180,E1 -28759.772,E2 -28759.772} C_VEL
LIN {X 0,Y 108.68,Z 303.139,A -85,B 0,C 180,E1 -28761.627,E2 -28761.627} C_VEL
LIN {X 0,Y 113.437,Z 289.056,A -85,B 0,C 180,E1 -28763.269,E2 -28763.269} C_VEL
LIN {X 0,Y 117.068,Z 274.439,A -85,B 0,C 180,E1 -28764.416,E2 -28764.416} C_VEL
LIN {X 0,Y 119.445,Z 260.082,A -85,B 0,C 180,E1 -28765.065,E2 -28765.065} C_VEL
LIN {X 0,Y 122.978,Z 227.035,A -85,B 0,C 180,E1 -28766.171,E2 -28766.171} C_VEL
LIN {X 0,Y 120.728,Z 220.999,A -85,B 0,C 180,E1 -28769.508,E2 -28769.508} C_VEL
LIN {X 0,Y 118.528,Z 215.802,A -85,B 0,C 180,E1 -28773.295,E2 -28773.295} C_VEL
LIN {X 0,Y 116.463,Z 211.317,A -85,B 0,C 180,E1 -28777.796,E2 -28777.796} C_VEL
LIN {X 0,Y 115.036,Z 208.17,A -85,B 0,C 180,E1 -28782.226,E2 -28782.226} C_VEL
LIN {X 0,Y 113.964,Z 204.393,A -85,B 0,C 180,E1 -28791.454,E2 -28791.454} C_VEL
LIN {X 0,Y 114.055,Z 204.198,A -85,B 0,C 180,E1 -28793.838,E2 -28793.838} C_VEL
LIN {X 0,Y 114.828,Z 207.45,A -85,B 0,C 180,E1 -28800.452,E2 -28800.452} C_VEL
LIN {X 0,Y 115.347,Z 208.5,A -85,B 0,C 180,E1 -28802.418,E2 -28802.418} C_VEL
LIN {X 0,Y 117.019,Z 212.281,A -85,B 0,C 180,E1 -28807.127,E2 -28807.127} C_VEL
LIN {X 0,Y 119.139,Z 217.071,A -85,B 0,C 180,E1 -28811.428,E2 -28811.428} C_VEL
LIN {X 0,Y 121.67,Z 223.45,A -85,B 0,C 180,E1 -28815.573,E2 -28815.573} C_VEL
LIN {X 0,Y 123.048,Z 227.646,A -85,B 0,C 180,E1 -28817.62,E2 -28817.62} C_VEL
LIN {X 0,Y 118.7,Z 267.828,A -85,B 0,C 180,E1 -28819.031,E2 -28819.031} C_VEL
LIN {X 0,Y 115.803,Z 282.617,A -85,B 0,C 180,E1 -28819.858,E2 -28819.858} C_VEL
LIN {X 0,Y 111.579,Z 297.269,A -85,B 0,C 180,E1 -28821.109,E2 -28821.109} C_VEL
LIN {X 0,Y 106.606,Z 310.217,A -85,B 0,C 180,E1 -28822.654,E2 -28822.654} C_VEL
LIN {X 0,Y 100.387,Z 323.246,A -85,B 0,C 180,E1 -28824.852,E2 -28824.852} C_VEL
LIN {X 0,Y 94.094,Z 334.332,A -85,B 0,C 180,E1 -28827.521,E2 -28827.521} C_VEL
LIN {X 0,Y 88.534,Z 342.922,A -85,B 0,C 180,E1 -28830.327,E2 -28830.327} C_VEL
LIN {X 0,Y 81.204,Z 352.908,A -85,B 0,C 180,E1 -28834.708,E2 -28834.708} C_VEL
LIN {X 0,Y 73.924,Z 361.964,A -85,B 0,C 180,E1 -28840.498,E2 -28840.498} C_VEL
LIN {X 0,Y 66.898,Z 370.176,A -85,B 0,C 180,E1 -28848.21,E2 -28848.21} C_VEL
LIN {X 0,Y 60.836,Z 377.553,A -85,B 0,C 180,E1 -28858.688,E2 -28858.688} C_VEL
LIN {X 0,Y 57.453,Z 382.297,A -85,B 0,C 180,E1 -28868.481,E2 -28868.481} C_VEL
LIN {X 0,Y 55.769,Z 386.108,A -85,B 0,C 180,E1 -28879.114,E2 -28879.114} C_VEL
LIN {X 0,Y 55.528,Z 389.019,A -85,B 0,C 180,E1 -28890.01,E2 -28890.01} C_VEL
LIN {X 0,Y 55.586,Z 390.458,A -85,B 0,C 180,E1 -28897.274,E2 -28897.274} C_VEL
LIN {X 0,Y 57.671,Z 392.296,A -85,B 0,C 180,E1 -28911.455,E2 -28911.455} C_VEL
LIN {X 0,Y 62.736,Z 392.835,A -85,B 0,C 180,E1 -28924.075,E2 -28924.075} C_VEL
LIN {X 0,Y 70.363,Z 392.1,A -85,B 0,C 180,E1 -28934.372,E2 -28934.372} C_VEL
LIN {X 0,Y 79.762,Z 390.085,A -85,B 0,C 180,E1 -28942.479,E2 -28942.479} C_VEL
LIN {X 0,Y 90.444,Z 386.736,A -85,B 0,C 180,E1 -28948.744,E2 -28948.744} C_VEL
LIN {X 0,Y 102.026,Z 381.955,A -85,B 0,C 180,E1 -28953.584,E2 -28953.584} C_VEL
LIN {X 0,Y 114.287,Z 375.594,A -85,B 0,C 180,E1 -28957.294,E2 -28957.294} C_VEL
LIN {X 0,Y 125.363,Z 368.553,A -85,B 0,C 180,E1 -28959.901,E2 -28959.901} C_VEL
LIN {X 0,Y 134.963,Z 361.244,A -85,B 0,C 180,E1 -28961.881,E2 -28961.881} C_VEL
LIN {X 0,Y 144.793,Z 352.479,A -85,B 0,C 180,E1 -28963.475,E2 -28963.475} C_VEL
LIN {X 0,Y 154.741,Z 341.894,A -85,B 0,C 180,E1 -28964.837,E2 -28964.837} C_VEL
LIN {X 0,Y 163.065,Z 331.252,A -85,B 0,C 180,E1 -28965.881,E2 -28965.881} C_VEL
LIN {X 0,Y 170.662,Z 319.621,A -85,B 0,C 180,E1 -28966.643,E2 -28966.643} C_VEL
LIN {X 0,Y 177.414,Z 306.875,A -85,B 0,C 180,E1 -28967.299,E2 -28967.299} C_VEL
LIN {X 0,Y 182.677,Z 294.314,A -85,B 0,C 180,E1 -28967.752,E2 -28967.752} C_VEL
LIN {X 0,Y 186.877,Z 281.155,A -85,B 0,C 180,E1 -28968.088,E2 -28968.088} C_VEL
LIN {X 0,Y 186.923,Z 280.76,A -85,B 0,C 180,E1 -28968.357,E2 -28968.357} C_VEL
LIN {X 0,Y 186.919,Z 278.816,A -85,B 0,C 180,E1 -28972.431,E2 -28972.431} C_VEL
LIN {X 0,Y 186.938,Z 279.038,A -85,B 0,C 180,E1 -28973.788,E2 -28973.788} C_VEL
LIN {X 0,Y 186.912,Z 280.196,A -85,B 0,C 180,E1 -28975.81,E2 -28975.81} C_VEL
LIN {X 0,Y 186.734,Z 281.068,A -85,B 0,C 180,E1 -28976.146,E2 -28976.146} C_VEL
LIN {X 0,Y 186.048,Z 283.546,A -85,B 0,C 180,E1 -28976.31,E2 -28976.31} C_VEL
LIN {X 0,Y 184.912,Z 287.043,A -85,B 0,C 180,E1 -28976.069,E2 -28976.069} C_VEL
LIN {X 0,Y 181.717,Z 295.442,A -85,B 0,C 180,E1 -28974.877,E2 -28974.877} C_VEL
LIN {X 0,Y 180.149,Z 299.224,A -85,B 0,C 180,E1 -28974.689,E2 -28974.689} C_VEL
LIN {X 0,Y 179.822,Z 299.969,A -85,B 0,C 180,E1 -28974.71,E2 -28974.71} C_VEL
LIN {X 0,Y 173.595,Z 312.944,A -85,B 0,C 180,E1 -28975.348,E2 -28975.348} C_VEL
LIN {X 0,Y 166.433,Z 324.886,A -85,B 0,C 180,E1 -28976.088,E2 -28976.088} C_VEL
LIN {X 0,Y 158.352,Z 335.967,A -85,B 0,C 180,E1 -28977.004,E2 -28977.004} C_VEL
LIN {X 0,Y 149.437,Z 346.145,A -85,B 0,C 180,E1 -28978.085,E2 -28978.085} C_VEL
LIN {X 0,Y 139.321,Z 355.8,A -85,B 0,C 180,E1 -28979.54,E2 -28979.54} C_VEL
LIN {X 0,Y 128.308,Z 364.535,A -85,B 0,C 180,E1 -28981.39,E2 -28981.39} C_VEL
LIN {X 0,Y 118.322,Z 371.13,A -85,B 0,C 180,E1 -28983.394,E2 -28983.394} C_VEL
LIN {X 0,Y 106.101,Z 377.788,A -85,B 0,C 180,E1 -28986.451,E2 -28986.451} C_VEL
LIN {X 0,Y 96.234,Z 382.116,A -85,B 0,C 180,E1 -28989.595,E2 -28989.595} C_VEL
LIN {X 0,Y 84.607,Z 386.118,A -85,B 0,C 180,E1 -28994.414,E2 -28994.414} C_VEL
LIN {X 0,Y 74.796,Z 388.562,A -85,B 0,C 180,E1 -28999.991,E2 -28999.991} C_VEL
LIN {X 0,Y 64.201,Z 390.139,A -85,B 0,C 180,E1 -29008.848,E2 -29008.848} C_VEL
LIN {X 0,Y 55.624,Z 390.266,A -85,B 0,C 180,E1 -29020.689,E2 -29020.689} C_VEL
LIN {X 0,Y 49.943,Z 388.96,A -85,B 0,C 180,E1 -29035.731,E2 -29035.731} C_VEL
LIN {X 0,Y 48.425,Z 387.761,A -85,B 0,C 180,E1 -29044.177,E2 -29044.177} C_VEL
LIN {X 0,Y 47.753,Z 386.194,A -85,B 0,C 180,E1 -29052.869,E2 -29052.869} C_VEL
LIN {X 0,Y 49.3,Z 381.928,A -85,B 0,C 180,E1 -29069.988,E2 -29069.988} C_VEL
LIN {X 0,Y 52.398,Z 377.755,A -85,B 0,C 180,E1 -29081.595,E2 -29081.595} C_VEL
LIN {X 0,Y 56.997,Z 372.57,A -85,B 0,C 180,E1 -29091.7,E2 -29091.7} C_VEL
LIN {X 0,Y 64.133,Z 365.162,A -85,B 0,C 180,E1 -29101.357,E2 -29101.357} C_VEL
LIN {X 0,Y 71.831,Z 356.755,A -85,B 0,C 180,E1 -29108.521,E2 -29108.521} C_VEL
LIN {X 0,Y 78.954,Z 348.122,A -85,B 0,C 180,E1 -29113.608,E2 -29113.608} C_VEL
LIN {X 0,Y 86.491,Z 337.868,A -85,B 0,C 180,E1 -29117.846,E2 -29117.846} C_VEL
LIN {X 0,Y 93.81,Z 326.503,A -85,B 0,C 180,E1 -29121.001,E2 -29121.001} C_VEL
LIN {X 0,Y 100.601,Z 313.918,A -85,B 0,C 180,E1 -29123.445,E2 -29123.445} C_VEL
LIN {X 0,Y 105.962,Z 301.769,A -85,B 0,C 180,E1 -29125.153,E2 -29125.153} C_VEL
LIN {X 0,Y 110.691,Z 287.896,A -85,B 0,C 180,E1 -29126.624,E2 -29126.624} C_VEL
LIN {X 0,Y 114.154,Z 274.086,A -85,B 0,C 180,E1 -29127.617,E2 -29127.617} C_VEL
LIN {X 0,Y 116.545,Z 259.825,A -85,B 0,C 180,E1 -29128.199,E2 -29128.199} C_VEL
LIN {X 0,Y 119.808,Z 230.301,A -85,B 0,C 180,E1 -29129.111,E2 -29129.111} C_VEL
LIN {X 0,Y 117.872,Z 224.781,A -85,B 0,C 180,E1 -29132.527,E2 -29132.527} C_VEL
LIN {X 0,Y 116.145,Z 220.475,A -85,B 0,C 180,E1 -29136.147,E2 -29136.147} C_VEL
LIN {X 0,Y 114.97,Z 217.741,A -85,B 0,C 180,E1 -29139.211,E2 -29139.211} C_VEL
LIN {X 0,Y 113.939,Z 215.077,A -85,B 0,C 180,E1 -29142.913,E2 -29142.913} C_VEL
LIN {X 0,Y 113.13,Z 211.166,A -85,B 0,C 180,E1 -29152.875,E2 -29152.875} C_VEL
LIN {X 0,Y 114.12,Z 215.188,A -85,B 0,C 180,E1 -29161.342,E2 -29161.342} C_VEL
LIN {X 0,Y 115.661,Z 219.088,A -85,B 0,C 180,E1 -29166.235,E2 -29166.235} C_VEL
LIN {X 0,Y 117.757,Z 224.546,A -85,B 0,C 180,E1 -29170.888,E2 -29170.888} C_VEL
LIN {X 0,Y 119.525,Z 229.483,A -85,B 0,C 180,E1 -29174.048,E2 -29174.048} C_VEL
LIN {X 0,Y 119.926,Z 230.695,A -85,B 0,C 180,E1 -29174.714,E2 -29174.714} C_VEL
LIN {X 0,Y 115.528,Z 268.882,A -85,B 0,C 180,E1 -29175.952,E2 -29175.952} C_VEL
LIN {X 0,Y 112.468,Z 283.489,A -85,B 0,C 180,E1 -29176.72,E2 -29176.72} C_VEL
LIN {X 0,Y 108.408,Z 297.023,A -85,B 0,C 180,E1 -29177.809,E2 -29177.809} C_VEL
LIN {X 0,Y 103.272,Z 309.984,A -85,B 0,C 180,E1 -29179.242,E2 -29179.242} C_VEL
LIN {X 0,Y 96.869,Z 322.939,A -85,B 0,C 180,E1 -29181.284,E2 -29181.284} C_VEL
LIN {X 0,Y 90.254,Z 334.111,A -85,B 0,C 180,E1 -29183.817,E2 -29183.817} C_VEL
LIN {X 0,Y 84.407,Z 342.703,A -85,B 0,C 180,E1 -29186.498,E2 -29186.498} C_VEL
LIN {X 0,Y 75.975,Z 353.521,A -85,B 0,C 180,E1 -29191.182,E2 -29191.182} C_VEL
LIN {X 0,Y 68.24,Z 362.444,A -85,B 0,C 180,E1 -29197.059,E2 -29197.059} C_VEL
LIN {X 0,Y 60.32,Z 370.972,A -85,B 0,C 180,E1 -29205.661,E2 -29205.661} C_VEL
LIN {X 0,Y 54.85,Z 376.888,A -85,B 0,C 180,E1 -29214.802,E2 -29214.802} C_VEL
LIN {X 0,Y 50.877,Z 381.733,A -85,B 0,C 180,E1 -29225.53,E2 -29225.53} C_VEL
LIN {X 0,Y 48.797,Z 385.638,A -85,B 0,C 180,E1 -29237.536,E2 -29237.536} C_VEL
LIN {X 0,Y 48.445,Z 388.596,A -85,B 0,C 180,E1 -29250.012,E2 -29250.012} C_VEL
LIN {X 0,Y 48.553,Z 390.076,A -85,B 0,C 180,E1 -29258.335,E2 -29258.335} C_VEL
LIN {X 0,Y 51.086,Z 391.999,A -85,B 0,C 180,E1 -29274.387,E2 -29274.387} C_VEL
LIN {X 0,Y 56.957,Z 392.623,A -85,B 0,C 180,E1 -29288.107,E2 -29288.107} C_VEL
LIN {X 0,Y 65.443,Z 391.98,A -85,B 0,C 180,E1 -29298.754,E2 -29298.754} C_VEL
LIN {X 0,Y 75.63,Z 390.064,A -85,B 0,C 180,E1 -29306.768,E2 -29306.768} C_VEL
LIN {X 0,Y 86.969,Z 386.824,A -85,B 0,C 180,E1 -29312.751,E2 -29312.751} C_VEL
LIN {X 0,Y 99.065,Z 382.148,A -85,B 0,C 180,E1 -29317.273,E2 -29317.273} C_VEL
LIN {X 0,Y 111.746,Z 375.89,A -85,B 0,C 180,E1 -29320.644,E2 -29320.644} C_VEL
LIN {X 0,Y 123.104,Z 368.967,A -85,B 0,C 180,E1 -29323.006,E2 -29323.006} C_VEL
LIN {X 0,Y 134.593,Z 360.441,A -85,B 0,C 180,E1 -29325.033,E2 -29325.033} C_VEL
LIN {X 0,Y 144.631,Z 351.55,A -85,B 0,C 180,E1 -29326.39,E2 -29326.39} C_VEL
LIN {X 0,Y 154.73,Z 340.828,A -85,B 0,C 180,E1 -29327.584,E2 -29327.584} C_VEL
LIN {X 0,Y 163.199,Z 329.999,A -85,B 0,C 180,E1 -29328.453,E2 -29328.453} C_VEL
LIN {X 0,Y 170.876,Z 318.154,A -85,B 0,C 180,E1 -29329.116,E2 -29329.116} C_VEL
LIN {X 0,Y 177.721,Z 305.064,A -85,B 0,C 180,E1 -29329.652,E2 -29329.652} C_VEL
LIN {X 0,Y 182.867,Z 292.509,A -85,B 0,C 180,E1 -29330.021,E2 -29330.021} C_VEL
LIN {X 0,Y 184.42,Z 287.895,A -85,B 0,C 180,E1 -29330.123,E2 -29330.123} C_VEL
LIN {X 0,Y 184.781,Z 286.767,A -85,B 0,C 180,E1 -29330.27,E2 -29330.27} C_VEL
LIN {X 0,Y 184.969,Z 285.772,A -85,B 0,C 180,E1 -29333.448,E2 -29333.448} C_VEL
LIN {X 0,Y 184.897,Z 286.204,A -85,B 0,C 180,E1 -29334.209,E2 -29334.209} C_VEL
LIN {X 0,Y 180.284,Z 298.91,A -85,B 0,C 180,E1 -29334.664,E2 -29334.664} C_VEL
LIN {X 0,Y 179.822,Z 299.969,A -85,B 0,C 180,E1 -29334.71,E2 -29334.71} C_VEL
LIN {X 0,Y 177.357,Z 305.465,A -85,B 0,C 180,E1 -29334.743,E2 -29334.743} C_VEL
LIN {X 0,Y 172.784,Z 314.179,A -85,B 0,C 180,E1 -29334.23,E2 -29334.23} C_VEL
LIN {X 0,Y 167.787,Z 322.509,A -85,B 0,C 180,E1 -29333.715,E2 -29333.715} C_VEL
LIN {X 0,Y 164.532,Z 327.329,A -85,B 0,C 180,E1 -29333.764,E2 -29333.764} C_VEL
LIN {X 0,Y 156.196,Z 338.216,A -85,B 0,C 180,E1 -29334.601,E2 -29334.601} C_VEL
LIN {X 0,Y 146.263,Z 348.961,A -85,B 0,C 180,E1 -29335.64,E2 -29335.64} C_VEL
LIN {X 0,Y 137.685,Z 356.735,A -85,B 0,C 180,E1 -29336.72,E2 -29336.72} C_VEL
LIN {X 0,Y 126.568,Z 365.268,A -85,B 0,C 180,E1 -29338.313,E2 -29338.313} C_VEL
LIN {X 0,Y 114.62,Z 372.793,A -85,B 0,C 180,E1 -29340.424,E2 -29340.424} C_VEL
LIN {X 0,Y 102.072,Z 379.11,A -85,B 0,C 180,E1 -29343.215,E2 -29343.215} C_VEL
LIN {X 0,Y 91.901,Z 383.223,A -85,B 0,C 180,E1 -29346.142,E2 -29346.142} C_VEL
LIN {X 0,Y 81.771,Z 386.412,A -85,B 0,C 180,E1 -29349.881,E2 -29349.881} C_VEL
LIN {X 0,Y 72.554,Z 388.597,A -85,B 0,C 180,E1 -29354.354,E2 -29354.354} C_VEL
LIN {X 0,Y 60.913,Z 390.273,A -85,B 0,C 180,E1 -29362.604,E2 -29362.604} C_VEL
LIN {X 0,Y 51.036,Z 390.498,A -85,B 0,C 180,E1 -29374.266,E2 -29374.266} C_VEL
LIN {X 0,Y 43.932,Z 389.29,A -85,B 0,C 180,E1 -29390.199,E2 -29390.199} C_VEL
LIN {X 0,Y 41.859,Z 388.147,A -85,B 0,C 180,E1 -29399.74,E2 -29399.74} C_VEL
LIN {X 0,Y 40.746,Z 386.652,A -85,B 0,C 180,E1 -29409.805,E2 -29409.805} C_VEL
LIN {X 0,Y 41.254,Z 383.666,A -85,B 0,C 180,E1 -29425.1,E2 -29425.1} C_VEL
LIN {X 0,Y 44.059,Z 379.846,A -85,B 0,C 180,E1 -29439.165,E2 -29439.165} C_VEL
LIN {X 0,Y 48.569,Z 375.136,A -85,B 0,C 180,E1 -29451.195,E2 -29451.195} C_VEL
LIN {X 0,Y 55.762,Z 368.285,A -85,B 0,C 180,E1 -29462.376,E2 -29462.376} C_VEL
LIN {X 0,Y 63.144,Z 361.127,A -85,B 0,C 180,E1 -29469.778,E2 -29469.778} C_VEL
LIN {X 0,Y 71.162,Z 352.541,A -85,B 0,C 180,E1 -29475.715,E2 -29475.715} C_VEL
LIN {X 0,Y 79.626,Z 342.167,A -85,B 0,C 180,E1 -29480.549,E2 -29480.549} C_VEL
LIN {X 0,Y 88.018,Z 330.468,A -85,B 0,C 180,E1 -29483.934,E2 -29483.934} C_VEL
LIN {X 0,Y 94.951,Z 318.821,A -85,B 0,C 180,E1 -29486.365,E2 -29486.365} C_VEL
LIN {X 0,Y 101.251,Z 306.007,A -85,B 0,C 180,E1 -29488.232,E2 -29488.232} C_VEL
LIN {X 0,Y 106.317,Z 292.891,A -85,B 0,C 180,E1 -29489.655,E2 -29489.655} C_VEL
LIN {X 0,Y 110.468,Z 278.709,A -85,B 0,C 180,E1 -29490.687,E2 -29490.687} C_VEL
LIN {X 0,Y 113.159,Z 265.247,A -85,B 0,C 180,E1 -29491.33,E2 -29491.33} C_VEL
LIN {X 0,Y 116.902,Z 233.63,A -85,B 0,C 180,E1 -29492.234,E2 -29492.234} C_VEL
LIN {X 0,Y 115.102,Z 228.224,A -85,B 0,C 180,E1 -29496.205,E2 -29496.205} C_VEL
LIN {X 0,Y 113.637,Z 224.312,A -85,B 0,C 180,E1 -29500.387,E2 -29500.387} C_VEL
LIN {X 0,Y 112.754,Z 221.8,A -85,B 0,C 180,E1 -29504.094,E2 -29504.094} C_VEL
LIN {X 0,Y 112.24,Z 218.251,A -85,B 0,C 180,E1 -29512.818,E2 -29512.818} C_VEL
LIN {X 0,Y 112.979,Z 222.012,A -85,B 0,C 180,E1 -29520.459,E2 -29520.459} C_VEL
LIN {X 0,Y 114.256,Z 225.698,A -85,B 0,C 180,E1 -29525.105,E2 -29525.105} C_VEL
LIN {X 0,Y 116.045,Z 230.944,A -85,B 0,C 180,E1 -29529.598,E2 -29529.598} C_VEL
LIN {X 0,Y 117.005,Z 233.957,A -85,B 0,C 180,E1 -29531.589,E2 -29531.589} C_VEL
LIN {X 0,Y 112.885,Z 268.579,A -85,B 0,C 180,E1 -29532.639,E2 -29532.639} C_VEL
LIN {X 0,Y 109.837,Z 282.894,A -85,B 0,C 180,E1 -29533.322,E2 -29533.322} C_VEL
LIN {X 0,Y 105.618,Z 296.663,A -85,B 0,C 180,E1 -29534.323,E2 -29534.323} C_VEL
LIN {X 0,Y 100.327,Z 309.662,A -85,B 0,C 180,E1 -29535.614,E2 -29535.614} C_VEL
LIN {X 0,Y 94.547,Z 321.125,A -85,B 0,C 180,E1 -29537.22,E2 -29537.22} C_VEL
LIN {X 0,Y 90.045,Z 328.876,A -85,B 0,C 180,E1 -29538.682,E2 -29538.682} C_VEL
LIN {X 0,Y 82.185,Z 340.442,A -85,B 0,C 180,E1 -29541.59,E2 -29541.59} C_VEL
LIN {X 0,Y 73.97,Z 350.792,A -85,B 0,C 180,E1 -29545.516,E2 -29545.516} C_VEL
LIN {X 0,Y 65.51,Z 360.14,A -85,B 0,C 180,E1 -29550.896,E2 -29550.896} C_VEL
LIN {X 0,Y 57.26,Z 368.32,A -85,B 0,C 180,E1 -29558.176,E2 -29558.176} C_VEL
LIN {X 0,Y 51.064,Z 374.355,A -85,B 0,C 180,E1 -29566.532,E2 -29566.532} C_VEL
LIN {X 0,Y 45.783,Z 379.626,A -85,B 0,C 180,E1 -29577.517,E2 -29577.517} C_VEL
LIN {X 0,Y 42.485,Z 383.903,A -85,B 0,C 180,E1 -29590.694,E2 -29590.694} C_VEL
LIN {X 0,Y 41.461,Z 386.233,A -85,B 0,C 180,E1 -29600.255,E2 -29600.255} C_VEL
LIN {X 0,Y 41.344,Z 388.165,A -85,B 0,C 180,E1 -29610.014,E2 -29610.014} C_VEL
LIN {X 0,Y 41.531,Z 389.687,A -85,B 0,C 180,E1 -29619.757,E2 -29619.757} C_VEL
LIN {X 0,Y 44.684,Z 391.692,A -85,B 0,C 180,E1 -29638.168,E2 -29638.168} C_VEL
LIN {X 0,Y 51.526,Z 392.404,A -85,B 0,C 180,E1 -29653.013,E2 -29653.013} C_VEL
LIN {X 0,Y 60.969,Z 391.849,A -85,B 0,C 180,E1 -29663.81,E2 -29663.81} C_VEL
LIN {X 0,Y 71.967,Z 390.021,A -85,B 0,C 180,E1 -29671.526,E2 -29671.526} C_VEL
LIN {X 0,Y 83.948,Z 386.878,A -85,B 0,C 180,E1 -29677.075,E2 -29677.075} C_VEL
LIN {X 0,Y 96.539,Z 382.33,A -85,B 0,C 180,E1 -29681.172,E2 -29681.172} C_VEL
LIN {X 0,Y 109.604,Z 376.187,A -85,B 0,C 180,E1 -29684.135,E2 -29684.135} C_VEL
LIN {X 0,Y 121.221,Z 369.379,A -85,B 0,C 180,E1 -29686.212,E2 -29686.212} C_VEL
LIN {X 0,Y 132.942,Z 360.982,A -85,B 0,C 180,E1 -29687.979,E2 -29687.979} C_VEL
LIN {X 0,Y 143.132,Z 352.239,A -85,B 0,C 180,E1 -29689.14,E2 -29689.14} C_VEL
LIN {X 0,Y 153.369,Z 341.691,A -85,B 0,C 180,E1 -29690.157,E2 -29690.157} C_VEL
LIN {X 0,Y 161.94,Z 331.07,A -85,B 0,C 180,E1 -29690.886,E2 -29690.886} C_VEL
LIN {X 0,Y 169.694,Z 319.493,A -85,B 0,C 180,E1 -29691.438,E2 -29691.438} C_VEL
LIN {X 0,Y 176.273,Z 307.449,A -85,B 0,C 180,E1 -29691.871,E2 -29691.871} C_VEL
LIN {X 0,Y 179.358,Z 300.747,A -85,B 0,C 180,E1 -29692.064,E2 -29692.064} C_VEL
LIN {X 0,Y 179.968,Z 299.334,A -85,B 0,C 180,E1 -29692.41,E2 -29692.41} C_VEL
LIN {X 0,Y 174.066,Z 311.754,A -85,B 0,C 180,E1 -29692.935,E2 -29692.935} C_VEL
LIN {X 0,Y 167.108,Z 323.522,A -85,B 0,C 180,E1 -29693.535,E2 -29693.535} C_VEL
LIN {X 0,Y 164.532,Z 327.329,A -85,B 0,C 180,E1 -29693.764,E2 -29693.764} C_VEL
LIN {X 0,Y 160.728,Z 332.652,A -85,B 0,C 180,E1 -29693.878,E2 -29693.878} C_VEL
LIN {X 0,Y 153.81,Z 341.101,A -85,B 0,C 180,E1 -29693.499,E2 -29693.499} C_VEL
LIN {X 0,Y 146.253,Z 348.96,A -85,B 0,C 180,E1 -29693.12,E2 -29693.12} C_VEL
LIN {X 0,Y 141.436,Z 353.355,A -85,B 0,C 180,E1 -29693.289,E2 -29693.289} C_VEL
LIN {X 0,Y 130.63,Z 362.157,A -85,B 0,C 180,E1 -29694.494,E2 -29694.494} C_VEL
LIN {X 0,Y 119.792,Z 369.476,A -85,B 0,C 180,E1 -29695.897,E2 -29695.897} C_VEL
LIN {X 0,Y 109.035,Z 375.48,A -85,B 0,C 180,E1 -29697.646,E2 -29697.646} C_VEL
LIN {X 0,Y 97.292,Z 380.816,A -85,B 0,C 180,E1 -29699.986,E2 -29699.986} C_VEL
LIN {X 0,Y 84.493,Z 385.321,A -85,B 0,C 180,E1 -29703.39,E2 -29703.39} C_VEL
LIN {X 0,Y 71.055,Z 388.632,A -85,B 0,C 180,E1 -29708.416,E2 -29708.416} C_VEL
LIN {X 0,Y 58.422,Z 390.407,A -85,B 0,C 180,E1 -29715.731,E2 -29715.731} C_VEL
LIN {X 0,Y 47.183,Z 390.731,A -85,B 0,C 180,E1 -29726.63,E2 -29726.63} C_VEL
LIN {X 0,Y 38.462,Z 389.619,A -85,B 0,C 180,E1 -29743.017,E2 -29743.017} C_VEL
LIN {X 0,Y 35.618,Z 388.523,A -85,B 0,C 180,E1 -29753.685,E2 -29753.685} C_VEL
LIN {X 0,Y 33.909,Z 387.075,A -85,B 0,C 180,E1 -29765.492,E2 -29765.492} C_VEL
LIN {X 0,Y 34.691,Z 383.067,A -85,B 0,C 180,E1 -29789.983,E2 -29789.983} C_VEL
LIN {X 0,Y 38.413,Z 379.005,A -85,B 0,C 180,E1 -29805.913,E2 -29805.913} C_VEL
LIN {X 0,Y 43.99,Z 374.03,A -85,B 0,C 180,E1 -29818.624,E2 -29818.624} C_VEL
LIN {X 0,Y 52.445,Z 366.866,A -85,B 0,C 180,E1 -29829.52,E2 -29829.52} C_VEL
LIN {X 0,Y 60.981,Z 359.07,A -85,B 0,C 180,E1 -29836.606,E2 -29836.606} C_VEL
LIN {X 0,Y 69.384,Z 350.4,A -85,B 0,C 180,E1 -29841.708,E2 -29841.708} C_VEL
LIN {X 0,Y 76.842,Z 341.532,A -85,B 0,C 180,E1 -29845.387,E2 -29845.387} C_VEL
LIN {X 0,Y 84.815,Z 330.844,A -85,B 0,C 180,E1 -29848.126,E2 -29848.126} C_VEL
LIN {X 0,Y 92.005,Z 319.237,A -85,B 0,C 180,E1 -29850.318,E2 -29850.318} C_VEL
LIN {X 0,Y 98.506,Z 306.475,A -85,B 0,C 180,E1 -29851.982,E2 -29851.982} C_VEL
LIN {X 0,Y 103.744,Z 293.39,A -85,B 0,C 180,E1 -29853.257,E2 -29853.257} C_VEL
LIN {X 0,Y 108.171,Z 278.71,A -85,B 0,C 180,E1 -29854.201,E2 -29854.201} C_VEL
LIN {X 0,Y 110.818,Z 265.807,A -85,B 0,C 180,E1 -29854.754,E2 -29854.754} C_VEL
LIN {X 0,Y 114.315,Z 237.234,A -85,B 0,C 180,E1 -29855.513,E2 -29855.513} C_VEL
LIN {X 0,Y 113.087,Z 233.109,A -85,B 0,C 180,E1 -29858.994,E2 -29858.994} C_VEL
LIN {X 0,Y 112.058,Z 230.041,A -85,B 0,C 180,E1 -29862.837,E2 -29862.837} C_VEL
LIN {X 0,Y 111.6,Z 228.459,A -85,B 0,C 180,E1 -29865.423,E2 -29865.423} C_VEL
LIN {X 0,Y 111.326,Z 225.523,A -85,B 0,C 180,E1 -29872.759,E2 -29872.759} C_VEL
LIN {X 0,Y 111.873,Z 228.848,A -85,B 0,C 180,E1 -29879.595,E2 -29879.595} C_VEL
LIN {X 0,Y 112.971,Z 232.485,A -85,B 0,C 180,E1 -29884.178,E2 -29884.178} C_VEL
LIN {X 0,Y 114.412,Z 237.521,A -85,B 0,C 180,E1 -29888.343,E2 -29888.343} C_VEL
LIN {X 0,Y 110.63,Z 268.296,A -85,B 0,C 180,E1 -29889.192,E2 -29889.192} C_VEL
LIN {X 0,Y 107.505,Z 282.647,A -85,B 0,C 180,E1 -29889.792,E2 -29889.792} C_VEL
LIN {X 0,Y 103.239,Z 296.269,A -85,B 0,C 180,E1 -29890.662,E2 -29890.662} C_VEL
LIN {X 0,Y 97.806,Z 309.31,A -85,B 0,C 180,E1 -29891.781,E2 -29891.781} C_VEL
LIN {X 0,Y 91.544,Z 321.339,A -85,B 0,C 180,E1 -29893.261,E2 -29893.261} C_VEL
LIN {X 0,Y 86.301,Z 329.972,A -85,B 0,C 180,E1 -29894.776,E2 -29894.776} C_VEL
LIN {X 0,Y 79.02,Z 340.154,A -85,B 0,C 180,E1 -29897.065,E2 -29897.065} C_VEL
LIN {X 0,Y 71.172,Z 349.666,A -85,B 0,C 180,E1 -29900.291,E2 -29900.291} C_VEL
LIN {X 0,Y 62.128,Z 359.192,A -85,B 0,C 180,E1 -29905.204,E2 -29905.204} C_VEL
LIN {X 0,Y 53.992,Z 366.793,A -85,B 0,C 180,E1 -29911.404,E2 -29911.404} C_VEL
LIN {X 0,Y 46.116,Z 373.607,A -85,B 0,C 180,E1 -29920.379,E2 -29920.379} C_VEL
LIN {X 0,Y 39.938,Z 378.986,A -85,B 0,C 180,E1 -29932.001,E2 -29932.001} C_VEL
LIN {X 0,Y 35.814,Z 383.365,A -85,B 0,C 180,E1 -29946.909,E2 -29946.909} C_VEL
LIN {X 0,Y 34.476,Z 385.746,A -85,B 0,C 180,E1 -29958.255,E2 -29958.255} C_VEL
LIN {X 0,Y 34.259,Z 387.727,A -85,B 0,C 180,E1 -29970.017,E2 -29970.017} C_VEL
LIN {X 0,Y 34.556,Z 389.293,A -85,B 0,C 180,E1 -29981.752,E2 -29981.752} C_VEL
LIN {X 0,Y 38.548,Z 391.386,A -85,B 0,C 180,E1 -30003.176,E2 -30003.176} C_VEL
LIN {X 0,Y 46.564,Z 392.186,A -85,B 0,C 180,E1 -30019.015,E2 -30019.015} C_VEL
LIN {X 0,Y 57.043,Z 391.719,A -85,B 0,C 180,E1 -30029.61,E2 -30029.61} C_VEL
LIN {X 0,Y 68.847,Z 389.978,A -85,B 0,C 180,E1 -30036.762,E2 -30036.762} C_VEL
LIN {X 0,Y 81.434,Z 386.927,A -85,B 0,C 180,E1 -30041.704,E2 -30041.704} C_VEL
LIN {X 0,Y 94.484,Z 382.477,A -85,B 0,C 180,E1 -30045.257,E2 -30045.257} C_VEL
LIN {X 0,Y 107.881,Z 376.482,A -85,B 0,C 180,E1 -30047.761,E2 -30047.761} C_VEL
LIN {X 0,Y 119.732,Z 369.79,A -85,B 0,C 180,E1 -30049.504,E2 -30049.504} C_VEL
LIN {X 0,Y 131.654,Z 361.522,A -85,B 0,C 180,E1 -30050.983,E2 -30050.983} C_VEL
LIN {X 0,Y 141.971,Z 352.927,A -85,B 0,C 180,E1 -30051.942,E2 -30051.942} C_VEL
LIN {X 0,Y 148.876,Z 346.22,A -85,B 0,C 180,E1 -30052.486,E2 -30052.486} C_VEL
LIN {X 0,Y 141.436,Z 353.355,A -85,B 0,C 180,E1 -30053.289,E2 -30053.289} C_VEL
LIN {X 0,Y 137.345,Z 356.858,A -85,B 0,C 180,E1 -30053.542,E2 -30053.542} C_VEL
LIN {X 0,Y 128.813,Z 363.446,A -85,B 0,C 180,E1 -30053.611,E2 -30053.611} C_VEL
LIN {X 0,Y 119.876,Z 369.429,A -85,B 0,C 180,E1 -30053.485,E2 -30053.485} C_VEL
LIN {X 0,Y 115.26,Z 372.157,A -85,B 0,C 180,E1 -30053.521,E2 -30053.521} C_VEL
LIN {X 0,Y 108.208,Z 375.863,A -85,B 0,C 180,E1 -30053.947,E2 -30053.947} C_VEL
LIN {X 0,Y 105.846,Z 376.98,A -85,B 0,C 180,E1 -30054.243,E2 -30054.243} C_VEL
LIN {X 0,Y 96.144,Z 381.174,A -85,B 0,C 180,E1 -30055.794,E2 -30055.794} C_VEL
LIN {X 0,Y 84.385,Z 385.2,A -85,B 0,C 180,E1 -30058.238,E2 -30058.238} C_VEL
LIN {X 0,Y 70.346,Z 388.649,A -85,B 0,C 180,E1 -30062.294,E2 -30062.294} C_VEL
LIN {X 0,Y 56.834,Z 390.542,A -85,B 0,C 180,E1 -30068.335,E2 -30068.335} C_VEL
LIN {X 0,Y 44.311,Z 390.964,A -85,B 0,C 180,E1 -30077.852,E2 -30077.852} C_VEL
LIN {X 0,Y 33.778,Z 389.949,A -85,B 0,C 180,E1 -30093.639,E2 -30093.639} C_VEL
LIN {X 0,Y 29.919,Z 388.9,A -85,B 0,C 180,E1 -30105.168,E2 -30105.168} C_VEL
LIN {X 0,Y 27.333,Z 387.499,A -85,B 0,C 180,E1 -30119.028,E2 -30119.028} C_VEL
LIN {X 0,Y 27.361,Z 383.595,A -85,B 0,C 180,E1 -30149.979,E2 -30149.979} C_VEL
LIN {X 0,Y 31.53,Z 379.623,A -85,B 0,C 180,E1 -30169.513,E2 -30169.513} C_VEL
LIN {X 0,Y 37.85,Z 374.757,A -85,B 0,C 180,E1 -30183.833,E2 -30183.833} C_VEL
LIN {X 0,Y 47.151,Z 367.713,A -85,B 0,C 180,E1 -30195.056,E2 -30195.056} C_VEL
LIN {X 0,Y 57.497,Z 358.992,A -85,B 0,C 180,E1 -30202.598,E2 -30202.598} C_VEL
LIN {X 0,Y 66.77,Z 349.905,A -85,B 0,C 180,E1 -30207.342,E2 -30207.342} C_VEL
LIN {X 0,Y 74.649,Z 340.895,A -85,B 0,C 180,E1 -30210.542,E2 -30210.542} C_VEL
LIN {X 0,Y 82.907,Z 330.047,A -85,B 0,C 180,E1 -30212.868,E2 -30212.868} C_VEL
LIN {X 0,Y 90.357,Z 318.219,A -85,B 0,C 180,E1 -30214.7,E2 -30214.7} C_VEL
LIN {X 0,Y 97.05,Z 305.167,A -85,B 0,C 180,E1 -30216.085,E2 -30216.085} C_VEL
LIN {X 0,Y 102.441,Z 291.591,A -85,B 0,C 180,E1 -30217.188,E2 -30217.188} C_VEL
LIN {X 0,Y 106.573,Z 277.526,A -85,B 0,C 180,E1 -30217.908,E2 -30217.908} C_VEL
LIN {X 0,Y 109.134,Z 264.892,A -85,B 0,C 180,E1 -30218.352,E2 -30218.352} C_VEL
LIN {X 0,Y 112.098,Z 241.08,A -85,B 0,C 180,E1 -30218.907,E2 -30218.907} C_VEL
LIN {X 0,Y 111.059,Z 237.244,A -85,B 0,C 180,E1 -30223.12,E2 -30223.12} C_VEL
LIN {X 0,Y 110.579,Z 235.311,A -85,B 0,C 180,E1 -30226.212,E2 -30226.212} C_VEL
LIN {X 0,Y 110.409,Z 232.816,A -85,B 0,C 180,E1 -30232.698,E2 -30232.698} C_VEL
LIN {X 0,Y 110.761,Z 235.57,A -85,B 0,C 180,E1 -30238.505,E2 -30238.505} C_VEL
LIN {X 0,Y 111.554,Z 238.759,A -85,B 0,C 180,E1 -30242.624,E2 -30242.624} C_VEL
LIN {X 0,Y 112.161,Z 241.361,A -85,B 0,C 180,E1 -30244.942,E2 -30244.942} C_VEL
LIN {X 0,Y 108.808,Z 267.913,A -85,B 0,C 180,E1 -30245.609,E2 -30245.609} C_VEL
LIN {X 0,Y 105.786,Z 281.723,A -85,B 0,C 180,E1 -30246.088,E2 -30246.088} C_VEL
LIN {X 0,Y 101.3,Z 295.874,A -85,B 0,C 180,E1 -30246.845,E2 -30246.845} C_VEL
LIN {X 0,Y 95.745,Z 308.958,A -85,B 0,C 180,E1 -30247.765,E2 -30247.765} C_VEL
LIN {X 0,Y 89.381,Z 320.909,A -85,B 0,C 180,E1 -30248.973,E2 -30248.973} C_VEL
LIN {X 0,Y 83.912,Z 329.668,A -85,B 0,C 180,E1 -30250.267,E2 -30250.267} C_VEL
LIN {X 0,Y 76.389,Z 339.867,A -85,B 0,C 180,E1 -30252.205,E2 -30252.205} C_VEL
LIN {X 0,Y 67.389,Z 350.256,A -85,B 0,C 180,E1 -30255.306,E2 -30255.306} C_VEL
LIN {X 0,Y 57.867,Z 359.63,A -85,B 0,C 180,E1 -30259.768,E2 -30259.768} C_VEL
LIN {X 0,Y 49.778,Z 366.629,A -85,B 0,C 180,E1 -30265.088,E2 -30265.088} C_VEL
LIN {X 0,Y 41.828,Z 372.854,A -85,B 0,C 180,E1 -30272.875,E2 -30272.875} C_VEL
LIN {X 0,Y 34.591,Z 378.346,A -85,B 0,C 180,E1 -30284.698,E2 -30284.698} C_VEL
LIN {X 0,Y 28.274,Z 384.084,A -85,B 0,C 180,E1 -30308.13,E2 -30308.13} C_VEL
LIN {X 0,Y 27.147,Z 387.287,A -85,B 0,C 180,E1 -30330.021,E2 -30330.021} C_VEL
LIN {X 0,Y 27.633,Z 388.899,A -85,B 0,C 180,E1 -30344.755,E2 -30344.755} C_VEL
LIN {X 0,Y 32.819,Z 391.08,A -85,B 0,C 180,E1 -30369.996,E2 -30369.996} C_VEL
LIN {X 0,Y 42.231,Z 391.967,A -85,B 0,C 180,E1 -30386.339,E2 -30386.339} C_VEL
LIN {X 0,Y 53.777,Z 391.587,A -85,B 0,C 180,E1 -30396.204,E2 -30396.204} C_VEL
LIN {X 0,Y 66.356,Z 389.936,A -85,B 0,C 180,E1 -30402.432,E2 -30402.432} C_VEL
LIN {X 0,Y 79.485,Z 386.975,A -85,B 0,C 180,E1 -30406.588,E2 -30406.588} C_VEL
LIN {X 0,Y 92.931,Z 382.62,A -85,B 0,C 180,E1 -30409.496,E2 -30409.496} C_VEL
LIN {X 0,Y 106.602,Z 376.74,A -85,B 0,C 180,E1 -30411.495,E2 -30411.495} C_VEL
LIN {X 0,Y 113.473,Z 373.168,A -85,B 0,C 180,E1 -30412.326,E2 -30412.326} C_VEL
LIN {X 0,Y 115.055,Z 372.231,A -85,B 0,C 180,E1 -30412.971,E2 -30412.971} C_VEL
LIN {X 0,Y 105.846,Z 376.98,A -85,B 0,C 180,E1 -30414.243,E2 -30414.243} C_VEL
LIN {X 0,Y 100.343,Z 379.466,A -85,B 0,C 180,E1 -30414.705,E2 -30414.705} C_VEL
LIN {X 0,Y 90.854,Z 383.127,A -85,B 0,C 180,E1 -30414.512,E2 -30414.512} C_VEL
LIN {X 0,Y 81.167,Z 386.172,A -85,B 0,C 180,E1 -30414.316,E2 -30414.316} C_VEL
LIN {X 0,Y 75.357,Z 387.586,A -85,B 0,C 180,E1 -30415.001,E2 -30415.001} C_VEL
LIN {X 0,Y 63.294,Z 389.835,A -85,B 0,C 180,E1 -30418.156,E2 -30418.156} C_VEL
LIN {X 0,Y 49.319,Z 391.116,A -85,B 0,C 180,E1 -30423.89,E2 -30423.89} C_VEL
LIN {X 0,Y 36.193,Z 390.918,A -85,B 0,C 180,E1 -30433.788,E2 -30433.788} C_VEL
LIN {X 0,Y 25.154,Z 389.279,A -85,B 0,C 180,E1 -30453.007,E2 -30453.007} C_VEL
LIN {X 0,Y 21.318,Z 387.922,A -85,B 0,C 180,E1 -30468.714,E2 -30468.714} C_VEL
LIN {X 0,Y 19.393,Z 385.227,A -85,B 0,C 180,E1 -30499.53,E2 -30499.53} C_VEL
LIN {X 0,Y 22.876,Z 381.64,A -85,B 0,C 180,E1 -30527.866,E2 -30527.866} C_VEL
LIN {X 0,Y 29.539,Z 377.155,A -85,B 0,C 180,E1 -30546.475,E2 -30546.475} C_VEL
LIN {X 0,Y 39.338,Z 370.679,A -85,B 0,C 180,E1 -30559.378,E2 -30559.378} C_VEL
LIN {X 0,Y 50.24,Z 362.628,A -85,B 0,C 180,E1 -30567.047,E2 -30567.047} C_VEL
LIN {X 0,Y 58.717,Z 355.313,A -85,B 0,C 180,E1 -30571.16,E2 -30571.16} C_VEL
LIN {X 0,Y 66.466,Z 347.713,A -85,B 0,C 180,E1 -30573.977,E2 -30573.977} C_VEL
LIN {X 0,Y 74.827,Z 338.233,A -85,B 0,C 180,E1 -30576.293,E2 -30576.293} C_VEL
LIN {X 0,Y 83.275,Z 326.79,A -85,B 0,C 180,E1 -30578.158,E2 -30578.158} C_VEL
LIN {X 0,Y 90.976,Z 314.086,A -85,B 0,C 180,E1 -30579.481,E2 -30579.481} C_VEL
LIN {X 0,Y 96.961,Z 301.789,A -85,B 0,C 180,E1 -30580.418,E2 -30580.418} C_VEL
LIN {X 0,Y 102.056,Z 288.278,A -85,B 0,C 180,E1 -30581.222,E2 -30581.222} C_VEL
LIN {X 0,Y 105.869,Z 274.404,A -85,B 0,C 180,E1 -30581.801,E2 -30581.801} C_VEL
LIN {X 0,Y 108.434,Z 260.179,A -85,B 0,C 180,E1 -30582.072,E2 -30582.072} C_VEL
LIN {X 0,Y 110.236,Z 245.401,A -85,B 0,C 180,E1 -30582.403,E2 -30582.403} C_VEL
LIN {X 0,Y 109.631,Z 242.347,A -85,B 0,C 180,E1 -30586.556,E2 -30586.556} C_VEL
LIN {X 0,Y 109.503,Z 240.025,A -85,B 0,C 180,E1 -30592.637,E2 -30592.637} C_VEL
LIN {X 0,Y 109.703,Z 242.322,A -85,B 0,C 180,E1 -30597.488,E2 -30597.488} C_VEL
LIN {X 0,Y 110.269,Z 245.33,A -85,B 0,C 180,E1 -30601.307,E2 -30601.307} C_VEL
LIN {X 0,Y 110.294,Z 245.499,A -85,B 0,C 180,E1 -30601.454,E2 -30601.454} C_VEL
LIN {X 0,Y 107.186,Z 268.794,A -85,B 0,C 180,E1 -30601.954,E2 -30601.954} C_VEL
LIN {X 0,Y 103.725,Z 283.633,A -85,B 0,C 180,E1 -30602.386,E2 -30602.386} C_VEL
LIN {X 0,Y 98.942,Z 297.774,A -85,B 0,C 180,E1 -30602.976,E2 -30602.976} C_VEL
LIN {X 0,Y 93.303,Z 310.376,A -85,B 0,C 180,E1 -30603.679,E2 -30603.679} C_VEL
LIN {X 0,Y 86.722,Z 322.188,A -85,B 0,C 180,E1 -30604.663,E2 -30604.663} C_VEL
LIN {X 0,Y 78.625,Z 334.118,A -85,B 0,C 180,E1 -30606.123,E2 -30606.123} C_VEL
LIN {X 0,Y 70.952,Z 343.587,A -85,B 0,C 180,E1 -30607.954,E2 -30607.954} C_VEL
LIN {X 0,Y 60.825,Z 354.13,A -85,B 0,C 180,E1 -30610.901,E2 -30610.901} C_VEL
LIN {X 0,Y 50.945,Z 362.816,A -85,B 0,C 180,E1 -30615.102,E2 -30615.102} C_VEL
LIN {X 0,Y 39.929,Z 371.078,A -85,B 0,C 180,E1 -30622.51,E2 -30622.51} C_VEL
LIN {X 0,Y 29.985,Z 377.704,A -85,B 0,C 180,E1 -30634.914,E2 -30634.914} C_VEL
LIN {X 0,Y 21.817,Z 383.547,A -85,B 0,C 180,E1 -30661.136,E2 -30661.136} C_VEL
LIN {X 0,Y 20.039,Z 386.847,A -85,B 0,C 180,E1 -30690.029,E2 -30690.029} C_VEL
LIN {X 0,Y 20.848,Z 388.505,A -85,B 0,C 180,E1 -30709.73,E2 -30709.73} C_VEL
LIN {X 0,Y 27.733,Z 390.773,A -85,B 0,C 180,E1 -30739.517,E2 -30739.517} C_VEL
LIN {X 0,Y 38.737,Z 391.749,A -85,B 0,C 180,E1 -30755.148,E2 -30755.148} C_VEL
LIN {X 0,Y 51.311,Z 391.456,A -85,B 0,C 180,E1 -30763.53,E2 -30763.53} C_VEL
LIN {X 0,Y 64.562,Z 389.893,A -85,B 0,C 180,E1 -30768.483,E2 -30768.483} C_VEL
LIN {X 0,Y 78.141,Z 387.023,A -85,B 0,C 180,E1 -30771.674,E2 -30771.674} C_VEL
LIN {X 0,Y 85.003,Z 385.074,A -85,B 0,C 180,E1 -30772.866,E2 -30772.866} C_VEL
LIN {X 0,Y 84.956,Z 385.079,A -85,B 0,C 180,E1 -30773.125,E2 -30773.125} C_VEL
LIN {X 0,Y 75.357,Z 387.586,A -85,B 0,C 180,E1 -30775.001,E2 -30775.001} C_VEL
LIN {X 0,Y 69.442,Z 388.849,A -85,B 0,C 180,E1 -30775.827,E2 -30775.827} C_VEL
LIN {X 0,Y 59.294,Z 390.381,A -85,B 0,C 180,E1 -30775.879,E2 -30775.879} C_VEL
LIN {X 0,Y 51.118,Z 391.131,A -85,B 0,C 180,E1 -30775.821,E2 -30775.821} C_VEL
LIN {X 0,Y 45.064,Z 391.371,A -85,B 0,C 180,E1 -30776.779,E2 -30776.779} C_VEL
LIN {X 0,Y 43.106,Z 391.4,A -85,B 0,C 180,E1 -30777.504,E2 -30777.504} C_VEL
LIN {X 0,Y 35.166,Z 391.199,A -85,B 0,C 180,E1 -30781.744,E2 -30781.744} C_VEL
LIN {X 0,Y 21.975,Z 389.66,A -85,B 0,C 180,E1 -30796.278,E2 -30796.278} C_VEL
LIN {X 0,Y 16.461,Z 388.349,A -85,B 0,C 180,E1 -30811.298,E2 -30811.298} C_VEL
LIN {X 0,Y 12.221,Z 385.737,A -85,B 0,C 180,E1 -30853.24,E2 -30853.24} C_VEL
LIN {X 0,Y 16.094,Z 382.209,A -85,B 0,C 180,E1 -30895.852,E2 -30895.852} C_VEL
LIN {X 0,Y 24.154,Z 377.823,A -85,B 0,C 180,E1 -30916.635,E2 -30916.635} C_VEL
LIN {X 0,Y 35.107,Z 371.463,A -85,B 0,C 180,E1 -30928.266,E2 -30928.266} C_VEL
LIN {X 0,Y 46.738,Z 363.542,A -85,B 0,C 180,E1 -30934.422,E2 -30934.422} C_VEL
LIN {X 0,Y 55.646,Z 356.367,A -85,B 0,C 180,E1 -30937.567,E2 -30937.567} C_VEL
LIN {X 0,Y 65.365,Z 347.154,A -85,B 0,C 180,E1 -30940.158,E2 -30940.158} C_VEL
LIN {X 0,Y 73.121,Z 338.591,A -85,B 0,C 180,E1 -30941.62,E2 -30941.62} C_VEL
LIN {X 0,Y 81.761,Z 327.186,A -85,B 0,C 180,E1 -30942.97,E2 -30942.97} C_VEL
LIN {X 0,Y 89.599,Z 314.526,A -85,B 0,C 180,E1 -30943.895,E2 -30943.895} C_VEL
LIN {X 0,Y 95.683,Z 302.291,A -85,B 0,C 180,E1 -30944.566,E2 -30944.566} C_VEL
LIN {X 0,Y 100.857,Z 288.887,A -85,B 0,C 180,E1 -30945.181,E2 -30945.181} C_VEL
LIN {X 0,Y 104.821,Z 274.817,A -85,B 0,C 180,E1 -30945.617,E2 -30945.617} C_VEL
LIN {X 0,Y 107.359,Z 261.096,A -85,B 0,C 180,E1 -30945.803,E2 -30945.803} C_VEL
LIN {X 0,Y 108.741,Z 250.165,A -85,B 0,C 180,E1 -30946.003,E2 -30946.003} C_VEL
LIN {X 0,Y 108.564,Z 248.867,A -85,B 0,C 180,E1 -30948.335,E2 -30948.335} C_VEL
LIN {X 0,Y 108.591,Z 247.264,A -85,B 0,C 180,E1 -30952.575,E2 -30952.575} C_VEL
LIN {X 0,Y 108.686,Z 249.153,A -85,B 0,C 180,E1 -30956.552,E2 -30956.552} C_VEL
LIN {X 0,Y 108.794,Z 250.069,A -85,B 0,C 180,E1 -30957.855,E2 -30957.855} C_VEL
LIN {X 0,Y 106.043,Z 269.509,A -85,B 0,C 180,E1 -30958.188,E2 -30958.188} C_VEL
LIN {X 0,Y 102.655,Z 283.636,A -85,B 0,C 180,E1 -30958.487,E2 -30958.487} C_VEL
LIN {X 0,Y 97.96,Z 297.347,A -85,B 0,C 180,E1 -30958.89,E2 -30958.89} C_VEL
LIN {X 0,Y 92.238,Z 310.026,A -85,B 0,C 180,E1 -30959.353,E2 -30959.353} C_VEL
LIN {X 0,Y 85.467,Z 322.011,A -85,B 0,C 180,E1 -30960.015,E2 -30960.015} C_VEL
LIN {X 0,Y 77.309,Z 333.819,A -85,B 0,C 180,E1 -30961.003,E2 -30961.003} C_VEL
LIN {X 0,Y 68.575,Z 344.294,A -85,B 0,C 180,E1 -30962.438,E2 -30962.438} C_VEL
LIN {X 0,Y 58.153,Z 354.638,A -85,B 0,C 180,E1 -30964.534,E2 -30964.534} C_VEL
LIN {X 0,Y 47.686,Z 363.328,A -85,B 0,C 180,E1 -30967.73,E2 -30967.73} C_VEL
LIN {X 0,Y 36.116,Z 371.35,A -85,B 0,C 180,E1 -30973.421,E2 -30973.421} C_VEL
LIN {X 0,Y 26.542,Z 377.062,A -85,B 0,C 180,E1 -30982.122,E2 -30982.122} C_VEL
LIN {X 0,Y 15.939,Z 383.01,A -85,B 0,C 180,E1 -31008.64,E2 -31008.64} C_VEL
LIN {X 0,Y 12.945,Z 386.405,A -85,B 0,C 180,E1 -31050.044,E2 -31050.044} C_VEL
LIN {X 0,Y 14.351,Z 388.111,A -85,B 0,C 180,E1 -31079.367,E2 -31079.367} C_VEL
LIN {X 0,Y 23.733,Z 390.467,A -85,B 0,C 180,E1 -31112.724,E2 -31112.724} C_VEL
LIN {X 0,Y 36.323,Z 391.531,A -85,B 0,C 180,E1 -31125.398,E2 -31125.398} C_VEL
LIN {X 0,Y 49.76,Z 391.325,A -85,B 0,C 180,E1 -31131.44,E2 -31131.44} C_VEL
LIN {X 0,Y 52.621,Z 391.107,A -85,B 0,C 180,E1 -31132.3,E2 -31132.3} C_VEL
LIN {X 0,Y 49.388,Z 391.268,A -85,B 0,C 180,E1 -31135.069,E2 -31135.069} C_VEL
LIN {X 0,Y 43.106,Z 391.4,A -85,B 0,C 180,E1 -31137.504,E2 -31137.504} C_VEL
LIN {X 0,Y 37.353,Z 391.38,A -85,B 0,C 180,E1 -31139.389,E2 -31139.389} C_VEL
LIN {X 0,Y 27.481,Z 390.764,A -85,B 0,C 180,E1 -31140.455,E2 -31140.455} C_VEL
LIN {X 0,Y 19.569,Z 389.752,A -85,B 0,C 180,E1 -31141.277,E2 -31141.277} C_VEL
LIN {X 0,Y 13.826,Z 388.705,A -85,B 0,C 180,E1 -31145.217,E2 -31145.217} C_VEL
LIN {X 0,Y 12.026,Z 388.274,A -85,B 0,C 180,E1 -31148.421,E2 -31148.421} C_VEL
LIN {X 0,Y 5.314,Z 385.158,A -85,B 0,C 180,E1 -31229.892,E2 -31229.892} C_VEL
LIN {X 0,Y 13.234,Z 381.478,A -85,B 0,C 180,E1 -31282.734,E2 -31282.734} C_VEL
LIN {X 0,Y 23.3,Z 376.851,A -85,B 0,C 180,E1 -31294.749,E2 -31294.749} C_VEL
LIN {X 0,Y 35.392,Z 370.205,A -85,B 0,C 180,E1 -31300.554,E2 -31300.554} C_VEL
LIN {X 0,Y 47.625,Z 361.945,A -85,B 0,C 180,E1 -31303.533,E2 -31303.533} C_VEL
LIN {X 0,Y 58.083,Z 353.331,A -85,B 0,C 180,E1 -31305.423,E2 -31305.423} C_VEL
LIN {X 0,Y 68.535,Z 342.915,A -85,B 0,C 180,E1 -31306.913,E2 -31306.913} C_VEL
LIN {X 0,Y 77.356,Z 332.35,A -85,B 0,C 180,E1 -31307.563,E2 -31307.563} C_VEL
LIN {X 0,Y 85.247,Z 320.9,A -85,B 0,C 180,E1 -31308.204,E2 -31308.204} C_VEL
LIN {X 0,Y 92.276,Z 308.348,A -85,B 0,C 180,E1 -31308.66,E2 -31308.66} C_VEL
LIN {X 0,Y 97.96,Z 295.505,A -85,B 0,C 180,E1 -31309.077,E2 -31309.077} C_VEL
LIN {X 0,Y 102.456,Z 282.114,A -85,B 0,C 180,E1 -31309.397,E2 -31309.397} C_VEL
LIN {X 0,Y 105.676,Z 268.478,A -85,B 0,C 180,E1 -31309.555,E2 -31309.555} C_VEL
LIN {X 0,Y 107.528,Z 256.23,A -85,B 0,C 180,E1 -31309.622,E2 -31309.622} C_VEL
LIN {X 0,Y 107.609,Z 255.53,A -85,B 0,C 180,E1 -31309.735,E2 -31309.735} C_VEL
LIN {X 0,Y 107.682,Z 254.487,A -85,B 0,C 180,E1 -31312.512,E2 -31312.512} C_VEL
LIN {X 0,Y 107.67,Z 255.16,A -85,B 0,C 180,E1 -31314.198,E2 -31314.198} C_VEL
LIN {X 0,Y 105.261,Z 270.777,A -85,B 0,C 180,E1 -31314.385,E2 -31314.385} C_VEL
LIN {X 0,Y 101.554,Z 285.432,A -85,B 0,C 180,E1 -31314.58,E2 -31314.58} C_VEL
LIN {X 0,Y 96.584,Z 299.2,A -85,B 0,C 180,E1 -31314.793,E2 -31314.793} C_VEL
LIN {X 0,Y 90.733,Z 311.598,A -85,B 0,C 180,E1 -31314.993,E2 -31314.993} C_VEL
LIN {X 0,Y 83.666,Z 323.597,A -85,B 0,C 180,E1 -31315.296,E2 -31315.296} C_VEL
LIN {X 0,Y 76.63,Z 333.519,A -85,B 0,C 180,E1 -31315.749,E2 -31315.749} C_VEL
LIN {X 0,Y 68.647,Z 343.016,A -85,B 0,C 180,E1 -31316.416,E2 -31316.416} C_VEL
LIN {X 0,Y 58.027,Z 353.598,A -85,B 0,C 180,E1 -31317.463,E2 -31317.463} C_VEL
LIN {X 0,Y 47.26,Z 362.439,A -85,B 0,C 180,E1 -31319.038,E2 -31319.038} C_VEL
LIN {X 0,Y 35.15,Z 370.597,A -85,B 0,C 180,E1 -31321.967,E2 -31321.967} C_VEL
LIN {X 0,Y 24.751,Z 376.406,A -85,B 0,C 180,E1 -31326.576,E2 -31326.576} C_VEL
LIN {X 0,Y 14.698,Z 381.106,A -85,B 0,C 180,E1 -31337.136,E2 -31337.136} C_VEL
LIN {X 0,Y 6.58,Z 384.865,A -85,B 0,C 180,E1 -31377.825,E2 -31377.825} C_VEL
LIN {X 0,Y 5.841,Z 385.93,A -85,B 0,C 180,E1 -31410.098,E2 -31410.098} C_VEL
LIN {X 0,Y 8.871,Z 387.694,A -85,B 0,C 180,E1 -31462.497,E2 -31462.497} C_VEL
LIN {X 0,Y 21.421,Z 390.151,A -85,B 0,C 180,E1 -31489.978,E2 -31489.978} C_VEL
LIN {X 0,Y 24.483,Z 390.467,A -85,B 0,C 180,E1 -31494.01,E2 -31494.01} C_VEL
LIN {X 0,Y 12.026,Z 388.274,A -85,B 0,C 180,E1 -31508.421,E2 -31508.421} C_VEL
LIN {X 0,Y 9.892,Z 390.227,A -85,B 0,C 180,E1 -31514.533,E2 -31514.533} C_VEL
LIN {X 0,Y 9.892,Z 600,A -85,B 0,C 180,E1 -31514.533,E2 -31514.533} C_VEL
LIN {X 0,Y 9.892,Z 600,A -85,B 0,C 180,E1 -31514.533,E2 -31514.533}

QRS_NEXT_CUT()

QRS_NEXT()
QRS_HOME()

END
